                                        [[-16.4688,605.716,173],[0.880315,0.388416,0.250776,0.106249],[-1,2,-2,1],[5921.94,9E+09,9E+09,9E+09,9E+09,9E+09]],
                                        [[-16.4665,606.427,173.764],[0.879525,0.389144,0.251945,0.107365],[-1,2,-2,1],[5919.94,9E+09,9E+09,9E+09,9E+09,9E+09]],
                                        [[-16.4662,607.132,174.535],[0.878733,0.389877,0.253103,0.108461],[-1,2,-2,1],[5917.94,9E+09,9E+09,9E+09,9E+09,9E+09]],
                                        [[-16.463,607.837,175.307],[0.877932,0.390621,0.254258,0.109565],[-1,2,-2,1],[5915.94,9E+09,9E+09,9E+09,9E+09,9E+09]],
                                        [[-16.4608,608.535,176.077],[0.877129,0.391371,0.255402,0.11065],[-1,2,-2,1],[5913.94,9E+09,9E+09,9E+09,9E+09,9E+09]],
                                        [[-16.4544,609.233,176.846],[0.876338,0.392094,0.256543,0.111714],[-1,2,-2,1],[5911.94,9E+09,9E+09,9E+09,9E+09,9E+09]],
                                        [[-16.448,609.934,177.621],[0.875547,0.392822,0.25767,0.112755],[-1,2,-2,1],[5909.94,9E+09,9E+09,9E+09,9E+09,9E+09]],
                                        [[-16.4455,610.629,178.404],[0.874742,0.39359,0.25878,0.113781],[-1,2,-2,1],[5907.94,9E+09,9E+09,9E+09,9E+09,9E+09]],
                                        [[-16.4446,611.323,179.187],[0.873932,0.39437,0.259879,0.114795],[-1,2,-2,1],[5905.94,9E+09,9E+09,9E+09,9E+09,9E+09]],
                                        [[-16.4419,612.013,179.972],[0.87311,0.395177,0.260966,0.115802],[-1,2,-2,1],[5903.94,9E+09,9E+09,9E+09,9E+09,9E+09]],
                                        [[-16.4412,612.703,180.758],[0.872287,0.395996,0.262037,0.116783],[-1,2,-2,1],[5901.94,9E+09,9E+09,9E+09,9E+09,9E+09]],
                                        [[-16.4357,613.389,181.546],[0.871466,0.396828,0.263087,0.117726],[-1,2,-2,1],[5899.94,9E+09,9E+09,9E+09,9E+09,9E+09]],
                                        [[-16.4315,614.073,182.336],[0.870641,0.397685,0.264115,0.118634],[-1,2,-2,1],[5897.94,9E+09,9E+09,9E+09,9E+09,9E+09]],
                                        [[-16.4296,614.755,183.129],[0.869825,0.398544,0.26512,0.119495],[-1,2,-2,1],[5895.94,9E+09,9E+09,9E+09,9E+09,9E+09]],
                                        [[-16.4286,615.436,183.924],[0.869011,0.39942,0.2661,0.120308],[-1,2,-2,1],[5893.94,9E+09,9E+09,9E+09,9E+09,9E+09]],
                                        [[-16.4255,616.116,184.719],[0.868205,0.40029,0.267066,0.12109],[-1,2,-2,1],[5891.94,9E+09,9E+09,9E+09,9E+09,9E+09]],
                                        [[-16.4247,616.797,185.514],[0.867397,0.401171,0.268021,0.121861],[-1,2,-2,1],[5889.94,9E+09,9E+09,9E+09,9E+09,9E+09]],
                                        [[-16.426,617.481,186.317],[0.866592,0.402053,0.268962,0.122605],[-1,2,-2,1],[5887.94,9E+09,9E+09,9E+09,9E+09,9E+09]],
                                        [[-16.4241,618.163,187.124],[0.865786,0.402931,0.2699,0.123348],[-1,2,-2,1],[5885.94,9E+09,9E+09,9E+09,9E+09,9E+09]],
                                        [[-16.4169,618.844,187.93],[0.864989,0.403788,0.270837,0.124084],[-1,2,-2,1],[5883.94,9E+09,9E+09,9E+09,9E+09,9E+09]],
                                        [[-16.4138,619.522,188.739],[0.86419,0.40464,0.271774,0.124824],[-1,2,-2,1],[5881.94,9E+09,9E+09,9E+09,9E+09,9E+09]],
                                        [[-16.4083,620.197,189.55],[0.863399,0.405471,0.27271,0.125558],[-1,2,-2,1],[5879.94,9E+09,9E+09,9E+09,9E+09,9E+09]],
                                        [[-16.4046,620.865,190.357],[0.862604,0.406303,0.273645,0.126297],[-1,2,-2,1],[5877.94,9E+09,9E+09,9E+09,9E+09,9E+09]],
                                        [[-16.3968,621.534,191.171],[0.861814,0.407129,0.27457,0.127018],[-1,2,-2,1],[5875.94,9E+09,9E+09,9E+09,9E+09,9E+09]],
                                        [[-16.3905,622.204,191.985],[0.861029,0.407945,0.275491,0.127729],[-1,2,-2,1],[5873.94,9E+09,9E+09,9E+09,9E+09,9E+09]],
                                        [[-16.3854,622.872,192.8],[0.860247,0.408753,0.276409,0.128433],[-1,2,-2,1],[5871.94,9E+09,9E+09,9E+09,9E+09,9E+09]],
                                        [[-16.3832,623.539,193.617],[0.85946,0.409575,0.277314,0.129126],[-1,2,-2,1],[5869.94,9E+09,9E+09,9E+09,9E+09,9E+09]],
                                        [[-16.3782,624.203,194.438],[0.858671,0.410404,0.27821,0.129811],[-1,2,-2,1],[5867.94,9E+09,9E+09,9E+09,9E+09,9E+09]],
                                        [[-16.3702,624.868,195.256],[0.857885,0.411232,0.279098,0.130482],[-1,2,-2,1],[5865.94,9E+09,9E+09,9E+09,9E+09,9E+09]],
                                        [[-16.36,625.527,196.082],[0.857094,0.412086,0.279965,0.131129],[-1,2,-2,1],[5863.94,9E+09,9E+09,9E+09,9E+09,9E+09]],
                                        [[-16.3521,626.19,196.902],[0.856303,0.412944,0.280822,0.131761],[-1,2,-2,1],[5861.94,9E+09,9E+09,9E+09,9E+09,9E+09]],
                                        [[-16.343,626.851,197.732],[0.855501,0.413827,0.281667,0.132394],[-1,2,-2,1],[5859.94,9E+09,9E+09,9E+09,9E+09,9E+09]],
                                        [[-16.3373,627.513,198.562],[0.85469,0.414724,0.282507,0.133035],[-1,2,-2,1],[5857.94,9E+09,9E+09,9E+09,9E+09,9E+09]],
                                        [[-16.3314,628.172,199.395],[0.853875,0.415619,0.283348,0.133685],[-1,2,-2,1],[5855.94,9E+09,9E+09,9E+09,9E+09,9E+09]],
                                        [[-16.3256,628.826,200.223],[0.853047,0.416519,0.284196,0.134369],[-1,2,-2,1],[5853.94,9E+09,9E+09,9E+09,9E+09,9E+09]],
                                        [[-16.3209,629.482,201.058],[0.852211,0.417405,0.285059,0.135093],[-1,2,-2,1],[5851.94,9E+09,9E+09,9E+09,9E+09,9E+09]],
                                        [[-16.3138,630.136,201.895],[0.851373,0.418283,0.285926,0.135829],[-1,2,-2,1],[5849.94,9E+09,9E+09,9E+09,9E+09,9E+09]],
                                        [[-16.3061,630.787,202.736],[0.85053,0.419166,0.286788,0.136569],[-1,2,-2,1],[5847.94,9E+09,9E+09,9E+09,9E+09,9E+09]],
                                        [[-16.2994,631.434,203.573],[0.849683,0.420043,0.287654,0.137324],[-1,2,-2,1],[5845.94,9E+09,9E+09,9E+09,9E+09,9E+09]],
                                        [[-16.2926,632.082,204.418],[0.848835,0.420916,0.288519,0.138081],[-1,2,-2,1],[5843.94,9E+09,9E+09,9E+09,9E+09,9E+09]],
                                        [[-16.2844,632.728,205.265],[0.847968,0.421816,0.289378,0.138857],[-1,2,-2,1],[5841.94,9E+09,9E+09,9E+09,9E+09,9E+09]],
                                        [[-16.2779,633.376,206.114],[0.847102,0.422713,0.290233,0.139633],[-1,2,-2,1],[5839.94,9E+09,9E+09,9E+09,9E+09,9E+09]],
                                        [[-16.269,634.022,206.966],[0.846219,0.42363,0.291085,0.140426],[-1,2,-2,1],[5837.94,9E+09,9E+09,9E+09,9E+09,9E+09]],
                                        [[-16.254,634.668,207.827],[0.84534,0.42453,0.291941,0.141226],[-1,2,-2,1],[5835.94,9E+09,9E+09,9E+09,9E+09,9E+09]],
                                        [[-16.2422,635.309,208.683],[0.844451,0.425428,0.292804,0.142054],[-1,2,-2,1],[5833.94,9E+09,9E+09,9E+09,9E+09,9E+09]],
                                        [[-16.2264,635.948,209.541],[0.843559,0.426327,0.293663,0.142883],[-1,2,-2,1],[5831.94,9E+09,9E+09,9E+09,9E+09,9E+09]],
                                        [[-16.2095,636.584,210.4],[0.842667,0.427211,0.294528,0.143724],[-1,2,-2,1],[5829.94,9E+09,9E+09,9E+09,9E+09,9E+09]],
                                        [[-16.1954,637.216,211.261],[0.841771,0.428083,0.2954,0.144586],[-1,2,-2,1],[5827.94,9E+09,9E+09,9E+09,9E+09,9E+09]],
                                        [[-16.181,637.839,212.116],[0.840872,0.428941,0.296282,0.145471],[-1,2,-2,1],[5825.94,9E+09,9E+09,9E+09,9E+09,9E+09]],
                                        [[-16.1679,638.455,212.97],[0.83997,0.429778,0.297177,0.14638],[-1,2,-2,1],[5823.94,9E+09,9E+09,9E+09,9E+09,9E+09]],
                                        [[-16.1584,639.071,213.819],[0.839056,0.430609,0.298085,0.147329],[-1,2,-2,1],[5821.94,9E+09,9E+09,9E+09,9E+09,9E+09]],
                                        [[-16.1526,639.686,214.678],[0.838139,0.43142,0.299007,0.148306],[-1,2,-2,1],[5819.94,9E+09,9E+09,9E+09,9E+09,9E+09]],
                                        [[-16.1475,640.301,215.533],[0.837222,0.432196,0.299951,0.149319],[-1,2,-2,1],[5817.94,9E+09,9E+09,9E+09,9E+09,9E+09]],
                                        [[-16.1368,640.913,216.395],[0.836301,0.432942,0.300916,0.150368],[-1,2,-2,1],[5815.94,9E+09,9E+09,9E+09,9E+09,9E+09]],
                                        [[-16.1276,641.526,217.256],[0.83539,0.433649,0.301896,0.151431],[-1,2,-2,1],[5813.94,9E+09,9E+09,9E+09,9E+09,9E+09]],
                                        [[-16.1184,642.14,218.129],[0.834475,0.434361,0.302869,0.152488],[-1,2,-2,1],[5811.94,9E+09,9E+09,9E+09,9E+09,9E+09]],
                                        [[-16.1069,642.748,218.992],[0.833572,0.435048,0.303841,0.153532],[-1,2,-2,1],[5809.94,9E+09,9E+09,9E+09,9E+09,9E+09]],
                                        [[-16.0956,643.35,219.86],[0.832666,0.435728,0.304815,0.154583],[-1,2,-2,1],[5807.94,9E+09,9E+09,9E+09,9E+09,9E+09]],
                                        [[-16.0855,643.953,220.727],[0.831771,0.436383,0.305791,0.155625],[-1,2,-2,1],[5805.94,9E+09,9E+09,9E+09,9E+09,9E+09]],
                                        [[-16.0764,644.555,221.603],[0.83088,0.437017,0.306772,0.156671],[-1,2,-2,1],[5803.94,9E+09,9E+09,9E+09,9E+09,9E+09]],
                                        [[-16.0662,645.154,222.472],[0.829995,0.437631,0.307757,0.157714],[-1,2,-2,1],[5801.94,9E+09,9E+09,9E+09,9E+09,9E+09]],
                                        [[-16.0574,645.75,223.34],[0.829119,0.438233,0.308733,0.158737],[-1,2,-2,1],[5799.94,9E+09,9E+09,9E+09,9E+09,9E+09]],
                                        [[-16.0432,646.341,224.209],[0.828249,0.438818,0.309711,0.159754],[-1,2,-2,1],[5797.94,9E+09,9E+09,9E+09,9E+09,9E+09]],
                                        [[-16.0362,646.93,225.078],[0.827391,0.439394,0.310676,0.16074],[-1,2,-2,1],[5795.94,9E+09,9E+09,9E+09,9E+09,9E+09]],
                                        [[-16.0338,647.518,225.94],[0.826541,0.439972,0.311624,0.161694],[-1,2,-2,1],[5793.94,9E+09,9E+09,9E+09,9E+09,9E+09]],
                                        [[-16.0304,648.102,226.805],[0.825699,0.440542,0.312564,0.162627],[-1,2,-2,1],[5791.94,9E+09,9E+09,9E+09,9E+09,9E+09]],
                                        [[-16.029,648.686,227.678],[0.825273,0.441318,0.312417,0.162967],[-1,2,-2,1],[6236.68,9E+09,9E+09,9E+09,9E+09,9E+09]],
                                        [[-16.0274,649.267,228.552],[0.824444,0.441882,0.313339,0.163861],[-1,2,-2,1],[6236.68,9E+09,9E+09,9E+09,9E+09,9E+09]],
                                        [[-16.0246,649.849,229.427],[0.823612,0.442457,0.314251,0.164747],[-1,2,-2,1],[6236.68,9E+09,9E+09,9E+09,9E+09,9E+09]],
                                        [[-16.0245,650.432,230.308],[0.822787,0.443017,0.31516,0.165623],[-1,2,-2,1],[6236.68,9E+09,9E+09,9E+09,9E+09,9E+09]],
                                        [[-16.0238,651.022,231.193],[0.821962,0.44357,0.316071,0.166503],[-1,2,-2,1],[6236.68,9E+09,9E+09,9E+09,9E+09,9E+09]],
                                        [[-16.02,651.619,232.093],[0.821137,0.444132,0.316968,0.167366],[-1,2,-2,1],[6236.68,9E+09,9E+09,9E+09,9E+09,9E+09]],
                                        [[-16.0079,652.21,232.993],[0.820319,0.44469,0.317856,0.16821],[-1,2,-2,1],[6236.68,9E+09,9E+09,9E+09,9E+09,9E+09]],
                                        [[-15.9949,652.798,233.889],[0.819499,0.445255,0.318735,0.169047],[-1,2,-2,1],[6236.68,9E+09,9E+09,9E+09,9E+09,9E+09]],
                                        [[-15.9855,653.382,234.784],[0.818688,0.445811,0.319607,0.169866],[-1,2,-2,1],[6236.68,9E+09,9E+09,9E+09,9E+09,9E+09]],
                                        [[-15.9753,653.961,235.677],[0.817868,0.446388,0.320465,0.170679],[-1,2,-2,1],[6236.68,9E+09,9E+09,9E+09,9E+09,9E+09]],
                                        [[-15.9659,654.533,236.562],[0.817047,0.446969,0.321316,0.171487],[-1,2,-2,1],[6236.68,9E+09,9E+09,9E+09,9E+09,9E+09]],
                                        [[-15.9573,655.108,237.457],[0.816216,0.447577,0.322152,0.17229],[-1,2,-2,1],[6236.68,9E+09,9E+09,9E+09,9E+09,9E+09]],
                                        [[-15.9494,655.68,238.35],[0.815387,0.448182,0.322983,0.173087],[-1,2,-2,1],[6236.68,9E+09,9E+09,9E+09,9E+09,9E+09]],
                                        [[-15.9432,656.253,239.242],[0.985491,-0.093353,0.141246,-0.0119022],[-1,2,-2,1],[6236.68,9E+09,9E+09,9E+09,9E+09,9E+09]],
                                        [[-15.9337,656.818,240.132],[0.985491,-0.093353,0.141246,-0.0119022],[-1,2,-2,1],[6236.68,9E+09,9E+09,9E+09,9E+09,9E+09]],
                                        [[-15.9252,657.38,241.024],[0.985491,-0.093353,0.141246,-0.0119022],[-1,2,-2,1],[6236.68,9E+09,9E+09,9E+09,9E+09,9E+09]],
                                        [[-15.9178,657.942,241.917],[0.985491,-0.093353,0.141246,-0.0119022],[-1,2,-2,1],[6236.68,9E+09,9E+09,9E+09,9E+09,9E+09]],
                                        [[-15.9128,658.506,242.814],[0.985491,-0.093353,0.141246,-0.0119022],[-1,2,-2,1],[6236.68,9E+09,9E+09,9E+09,9E+09,9E+09]],
                                        [[-15.9043,659.069,243.712],[0.985491,-0.093353,0.141246,-0.0119022],[-1,2,-2,1],[6236.68,9E+09,9E+09,9E+09,9E+09,9E+09]],
                                        [[-15.8949,659.626,244.614],[0.985491,-0.093353,0.141246,-0.0119022],[-1,2,-2,1],[6236.68,9E+09,9E+09,9E+09,9E+09,9E+09]],
                                        [[-15.884,660.185,245.513],[0.985491,-0.093353,0.141246,-0.0119022],[-1,2,-2,1],[6236.68,9E+09,9E+09,9E+09,9E+09,9E+09]],
                                        [[-15.8746,660.737,246.412],[0.985491,-0.093353,0.141246,-0.0119022],[-1,2,-2,1],[6236.68,9E+09,9E+09,9E+09,9E+09,9E+09]],
                                        [[-15.864,661.292,247.315],[0.985491,-0.093353,0.141246,-0.0119022],[-1,2,-2,1],[6236.68,9E+09,9E+09,9E+09,9E+09,9E+09]],
                                        [[-15.8527,661.843,248.221],[0.985491,-0.093353,0.141246,-0.0119022],[-1,2,-2,1],[6236.68,9E+09,9E+09,9E+09,9E+09,9E+09]],
                                        [[-15.843,662.392,249.125],[0.985491,-0.093353,0.141246,-0.0119022],[-1,2,-2,1],[6236.68,9E+09,9E+09,9E+09,9E+09,9E+09]],
                                        [[-15.8348,662.938,250.028],[0.985491,-0.093353,0.141246,-0.0119022],[-1,2,-2,1],[6236.68,9E+09,9E+09,9E+09,9E+09,9E+09]],
                                        [[-15.8269,663.475,250.925],[0.985491,-0.093353,0.141246,-0.0119022],[-1,2,-2,1],[6236.68,9E+09,9E+09,9E+09,9E+09,9E+09]],
                                        [[-15.8195,664.012,251.826],[0.985491,-0.093353,0.141246,-0.0119022],[-1,2,-2,1],[6236.68,9E+09,9E+09,9E+09,9E+09,9E+09]],
                                        [[-15.8093,664.544,252.731],[0.985491,-0.093353,0.141246,-0.0119022],[-1,2,-2,1],[6236.68,9E+09,9E+09,9E+09,9E+09,9E+09]],
                                        [[-15.8028,665.078,253.634],[0.985491,-0.093353,0.141246,-0.0119022],[-1,2,-2,1],[6236.68,9E+09,9E+09,9E+09,9E+09,9E+09]],
                                        [[-15.7448,665.866,254.446],[0.985491,-0.093353,0.141246,-0.0119022],[-1,2,-2,1],[6236.68,9E+09,9E+09,9E+09,9E+09,9E+09]],
                                        [[-15.7745,666.532,255.443],[0.985491,-0.093353,0.141246,-0.0119022],[-1,2,-2,1],[6236.68,9E+09,9E+09,9E+09,9E+09,9E+09]],
                                        [[-15.687,666.936,256.291],[0.985491,-0.093353,0.141246,-0.0119022],[-1,2,-2,1],[6236.68,9E+09,9E+09,9E+09,9E+09,9E+09]],
                                        [[-15.7962,667.567,257.036],[0.985491,-0.093353,0.141246,-0.0119022],[-1,2,-2,1],[6236.68,9E+09,9E+09,9E+09,9E+09,9E+09]],
                                        [[-15.7655,667.961,257.997],[0.985491,-0.093353,0.141246,-0.0119022],[-1,2,-2,1],[6236.68,9E+09,9E+09,9E+09,9E+09,9E+09]],
                                        [[-15.7582,668.439,258.917],[0.985491,-0.093353,0.141246,-0.0119022],[-1,2,-2,1],[6236.68,9E+09,9E+09,9E+09,9E+09,9E+09]],
                                        [[-15.7515,668.992,259.752],[0.985491,-0.093353,0.141246,-0.0119022],[-1,2,-2,1],[6236.68,9E+09,9E+09,9E+09,9E+09,9E+09]],
                                        [[-15.7656,669.642,260.77],[0.985491,-0.093353,0.141246,-0.0119022],[-1,2,-2,1],[6236.68,9E+09,9E+09,9E+09,9E+09,9E+09]],
                                        [[-15.7587,670.18,261.601],[0.985491,-0.093353,0.141246,-0.0119022],[-1,2,-2,1],[6236.68,9E+09,9E+09,9E+09,9E+09,9E+09]],
                                        [[-15.7161,670.57,262.57],[0.985491,-0.093353,0.141246,-0.0119022],[-1,2,-2,1],[6236.68,9E+09,9E+09,9E+09,9E+09,9E+09]],
                                        [[-15.6787,671.123,263.369],[0.985491,-0.093353,0.141246,-0.0119022],[-1,2,-2,1],[6236.68,9E+09,9E+09,9E+09,9E+09,9E+09]],
                                        [[-15.6791,671.49,264.34],[0.985491,-0.093353,0.141246,-0.0119022],[-1,2,-2,1],[6236.68,9E+09,9E+09,9E+09,9E+09,9E+09]],
                                        [[-15.6649,672.148,265.426],[0.985491,-0.093353,0.141246,-0.0119022],[-1,2,-2,1],[6236.68,9E+09,9E+09,9E+09,9E+09,9E+09]],
                                        [[-15.6634,672.552,266.32],[0.985491,-0.093353,0.141246,-0.0119022],[-1,2,-2,1],[6236.68,9E+09,9E+09,9E+09,9E+09,9E+09]],
                                        [[-15.7081,673.113,267.156],[0.985491,-0.093353,0.141246,-0.0119022],[-1,2,-2,1],[6236.68,9E+09,9E+09,9E+09,9E+09,9E+09]],
                                        [[-15.8035,673.64,268.067],[0.985491,-0.093353,0.141246,-0.0119022],[-1,2,-2,1],[6236.68,9E+09,9E+09,9E+09,9E+09,9E+09]],
                                        [[-15.7371,674.137,269.037],[0.985491,-0.093353,0.141246,-0.0119022],[-1,2,-2,1],[6236.68,9E+09,9E+09,9E+09,9E+09,9E+09]],
                                        [[-15.6886,674.748,270.209],[0.985491,-0.093353,0.141246,-0.0119022],[-1,2,-2,1],[6236.68,9E+09,9E+09,9E+09,9E+09,9E+09]],
                                        [[-15.5399,675.156,271.121],[0.985491,-0.093353,0.141246,-0.0119022],[-1,2,-2,1],[6236.68,9E+09,9E+09,9E+09,9E+09,9E+09]],
                                        [[-15.6158,675.69,271.899],[0.985491,-0.093353,0.141246,-0.0119022],[-1,2,-2,1],[6236.68,9E+09,9E+09,9E+09,9E+09,9E+09]],
                                        [[-16.0685,673.406,268.406],[0.77744,0.463066,0.366155,0.216997],[-1,2,-2,1],[5666.45,9E+09,9E+09,9E+09,9E+09,9E+09]],
                                        [[-16.0667,673.912,269.336],[0.776504,0.463677,0.366854,0.21786],[-1,2,-2,1],[5664.45,9E+09,9E+09,9E+09,9E+09,9E+09]],
                                        [[-16.0608,674.413,270.268],[0.775562,0.4643,0.367544,0.218724],[-1,2,-2,1],[5662.45,9E+09,9E+09,9E+09,9E+09,9E+09]],
                                        [[-16.0574,674.912,271.2],[0.774624,0.464915,0.368232,0.219584],[-1,2,-2,1],[5660.45,9E+09,9E+09,9E+09,9E+09,9E+09]],
                                        [[-16.0531,675.409,272.134],[0.773684,0.465512,0.368929,0.220459],[-1,2,-2,1],[5658.45,9E+09,9E+09,9E+09,9E+09,9E+09]],
                                        [[-16.0517,675.907,273.069],[0.772745,0.466095,0.369632,0.221343],[-1,2,-2,1],[5656.45,9E+09,9E+09,9E+09,9E+09,9E+09]],
                                        [[-16.0519,676.4,274.005],[0.771804,0.466665,0.370342,0.222238],[-1,2,-2,1],[5654.45,9E+09,9E+09,9E+09,9E+09,9E+09]],
                                        [[-16.0514,676.893,274.944],[0.770864,0.467217,0.371059,0.223142],[-1,2,-2,1],[5652.45,9E+09,9E+09,9E+09,9E+09,9E+09]],
                                        [[-16.0469,677.385,275.881],[0.769911,0.467761,0.371788,0.224078],[-1,2,-2,1],[5650.45,9E+09,9E+09,9E+09,9E+09,9E+09]],
                                        [[-16.044,677.877,276.826],[0.768946,0.468304,0.372521,0.225035],[-1,2,-2,1],[5648.45,9E+09,9E+09,9E+09,9E+09,9E+09]],
                                        [[-16.0392,678.365,277.773],[0.767988,0.468831,0.373257,0.225989],[-1,2,-2,1],[5646.45,9E+09,9E+09,9E+09,9E+09,9E+09]],
                                        [[-16.036,678.849,278.717],[0.767021,0.469363,0.37399,0.226954],[-1,2,-2,1],[5644.45,9E+09,9E+09,9E+09,9E+09,9E+09]],
                                        [[-16.0322,679.333,279.659],[0.766051,0.469892,0.374724,0.227926],[-1,2,-2,1],[5642.45,9E+09,9E+09,9E+09,9E+09,9E+09]],
                                        [[-16.0278,679.812,280.606],[0.765079,0.470404,0.375466,0.228911],[-1,2,-2,1],[5640.45,9E+09,9E+09,9E+09,9E+09,9E+09]],
                                        [[-16.024,680.293,281.558],[0.764104,0.470915,0.376206,0.229898],[-1,2,-2,1],[5638.45,9E+09,9E+09,9E+09,9E+09,9E+09]],
                                        [[-16.0198,680.773,282.512],[0.763131,0.471429,0.376937,0.230878],[-1,2,-2,1],[5636.45,9E+09,9E+09,9E+09,9E+09,9E+09]],
                                        [[-16.0145,681.251,283.46],[0.762158,0.471947,0.37766,0.231851],[-1,2,-2,1],[5634.45,9E+09,9E+09,9E+09,9E+09,9E+09]],
                                        [[-16.0138,681.724,284.41],[0.761189,0.472469,0.378372,0.23281],[-1,2,-2,1],[5632.45,9E+09,9E+09,9E+09,9E+09,9E+09]],
                                        [[-16.0091,682.195,285.362],[0.760213,0.473002,0.379074,0.233769],[-1,2,-2,1],[5630.45,9E+09,9E+09,9E+09,9E+09,9E+09]],
                                        [[-16.0037,682.663,286.315],[0.759249,0.473515,0.379778,0.23472],[-1,2,-2,1],[5628.45,9E+09,9E+09,9E+09,9E+09,9E+09]],
                                        [[-16.0002,683.132,287.275],[0.758279,0.47404,0.380472,0.235671],[-1,2,-2,1],[5626.45,9E+09,9E+09,9E+09,9E+09,9E+09]],
                                        [[-15.9998,683.601,288.235],[0.75731,0.474559,0.381165,0.236619],[-1,2,-2,1],[5624.45,9E+09,9E+09,9E+09,9E+09,9E+09]],
                                        [[-15.9984,684.066,289.189],[0.756344,0.47506,0.381864,0.237573],[-1,2,-2,1],[5622.45,9E+09,9E+09,9E+09,9E+09,9E+09]],
                                        [[-15.9972,684.528,290.146],[0.755371,0.475548,0.382574,0.238549],[-1,2,-2,1],[5620.45,9E+09,9E+09,9E+09,9E+09,9E+09]],
                                        [[-15.9956,684.993,291.107],[0.754399,0.476012,0.383297,0.239538],[-1,2,-2,1],[5618.45,9E+09,9E+09,9E+09,9E+09,9E+09]],
                                        [[-15.9948,685.455,292.071],[0.753425,0.476466,0.384024,0.240534],[-1,2,-2,1],[5616.45,9E+09,9E+09,9E+09,9E+09,9E+09]],
                                        [[-15.9915,685.91,293.03],[0.752456,0.476913,0.384748,0.241522],[-1,2,-2,1],[5614.45,9E+09,9E+09,9E+09,9E+09,9E+09]],
                                        [[-15.9856,686.361,293.993],[0.751487,0.47735,0.385474,0.242515],[-1,2,-2,1],[5612.45,9E+09,9E+09,9E+09,9E+09,9E+09]],
                                        [[-15.9792,686.815,294.953],[0.750524,0.477787,0.386192,0.243494],[-1,2,-2,1],[5610.45,9E+09,9E+09,9E+09,9E+09,9E+09]],
                                        [[-15.9762,687.264,295.916],[0.749563,0.478218,0.386907,0.24447],[-1,2,-2,1],[5608.45,9E+09,9E+09,9E+09,9E+09,9E+09]],
                                        [[-15.9728,687.713,296.879],[0.748608,0.478635,0.387625,0.245442],[-1,2,-2,1],[5606.45,9E+09,9E+09,9E+09,9E+09,9E+09]],
                                        [[-15.9682,688.157,297.846],[0.747659,0.479026,0.388353,0.246418],[-1,2,-2,1],[5604.45,9E+09,9E+09,9E+09,9E+09,9E+09]],
                                        [[-15.9611,688.602,298.811],[0.746714,0.479407,0.389083,0.24739],[-1,2,-2,1],[5602.45,9E+09,9E+09,9E+09,9E+09,9E+09]],
                                        [[-15.9549,689.045,299.778],[0.74577,0.479767,0.389822,0.248372],[-1,2,-2,1],[5600.45,9E+09,9E+09,9E+09,9E+09,9E+09]],
                                        [[-15.9477,689.484,300.747],[0.744833,0.480109,0.390567,0.249351],[-1,2,-2,1],[5598.45,9E+09,9E+09,9E+09,9E+09,9E+09]],
                                        [[-15.9427,689.92,301.71],[0.743901,0.48041,0.391337,0.250347],[-1,2,-2,1],[5596.45,9E+09,9E+09,9E+09,9E+09,9E+09]],
                                        [[-15.937,690.355,302.679],[0.742968,0.480709,0.392103,0.25134],[-1,2,-2,1],[5594.45,9E+09,9E+09,9E+09,9E+09,9E+09]],
                                        [[-15.9339,690.788,303.649],[0.742046,0.480985,0.392876,0.252328],[-1,2,-2,1],[5592.45,9E+09,9E+09,9E+09,9E+09,9E+09]],
                                        [[-15.9298,691.221,304.618],[0.741122,0.481239,0.393663,0.253332],[-1,2,-2,1],[5590.45,9E+09,9E+09,9E+09,9E+09,9E+09]],
                                        [[-15.9293,691.655,305.587],[0.7402,0.481452,0.394477,0.254355],[-1,2,-2,1],[5588.45,9E+09,9E+09,9E+09,9E+09,9E+09]],
                                        [[-15.9292,692.085,306.557],[0.739277,0.481618,0.395323,0.255407],[-1,2,-2,1],[5586.45,9E+09,9E+09,9E+09,9E+09,9E+09]],
                                        [[-15.9263,692.514,307.521],[0.738364,0.481742,0.396191,0.256467],[-1,2,-2,1],[5584.45,9E+09,9E+09,9E+09,9E+09,9E+09]],
                                        [[-15.9216,692.941,308.493],[0.737456,0.481845,0.397069,0.257528],[-1,1,-2,1],[5582.45,9E+09,9E+09,9E+09,9E+09,9E+09]],
                                        [[-15.9172,693.363,309.467],[0.736562,0.481908,0.397964,0.258584],[-1,1,-2,1],[5580.45,9E+09,9E+09,9E+09,9E+09,9E+09]],
                                        [[-15.9142,693.788,310.44],[0.735675,0.481957,0.398862,0.259633],[-1,1,-2,1],[5578.45,9E+09,9E+09,9E+09,9E+09,9E+09]],
                                        [[-15.9086,694.206,311.41],[0.734792,0.482002,0.399755,0.260673],[-1,1,-2,1],[5576.45,9E+09,9E+09,9E+09,9E+09,9E+09]],
                                        [[-15.9037,694.623,312.379],[0.733929,0.482034,0.400641,0.261681],[-1,1,-2,1],[5574.45,9E+09,9E+09,9E+09,9E+09,9E+09]],
                                        [[-15.9004,695.04,313.347],[0.733084,0.482057,0.401521,0.26266],[-1,1,-2,1],[5572.45,9E+09,9E+09,9E+09,9E+09,9E+09]],
                                        [[-15.8998,695.464,314.319],[0.732249,0.482067,0.402399,0.263625],[-1,1,-2,1],[5570.45,9E+09,9E+09,9E+09,9E+09,9E+09]],
                                        [[-15.8966,695.882,315.293],[0.73142,0.482071,0.403274,0.264579],[-1,1,-2,1],[5568.45,9E+09,9E+09,9E+09,9E+09,9E+09]],
                                        [[-15.8968,696.298,316.268],[0.730612,0.482057,0.404147,0.265505],[-1,1,-2,1],[5566.45,9E+09,9E+09,9E+09,9E+09,9E+09]],
                                        [[-15.8962,696.712,317.237],[0.729816,0.48204,0.405011,0.266408],[-1,1,-2,1],[5564.45,9E+09,9E+09,9E+09,9E+09,9E+09]],
                                        [[-15.8968,697.124,318.204],[0.729028,0.482039,0.405853,0.267281],[-1,1,-2,1],[5562.45,9E+09,9E+09,9E+09,9E+09,9E+09]],
                                        [[-15.8945,697.536,319.179],[0.728241,0.482044,0.406688,0.26815],[-1,1,-2,1],[5560.45,9E+09,9E+09,9E+09,9E+09,9E+09]],
                                        [[-15.8941,697.946,320.155],[0.727464,0.482049,0.407512,0.268995],[-1,1,-2,1],[5558.45,9E+09,9E+09,9E+09,9E+09,9E+09]],
                                        [[-15.8962,698.36,321.128],[0.726692,0.482055,0.40833,0.26983],[-1,1,-2,1],[5556.45,9E+09,9E+09,9E+09,9E+09,9E+09]],
                                        [[-15.8976,698.773,322.102],[0.725921,0.482068,0.409138,0.270656],[-1,1,-2,1],[5554.45,9E+09,9E+09,9E+09,9E+09,9E+09]],
                                        [[-15.9029,699.184,323.07],[0.725166,0.482038,0.409968,0.271479],[-1,1,-2,1],[5552.45,9E+09,9E+09,9E+09,9E+09,9E+09]],
                                        [[-15.9034,699.593,324.039],[0.724399,0.482035,0.41078,0.272302],[-1,1,-2,1],[5550.45,9E+09,9E+09,9E+09,9E+09,9E+09]],
                                        [[-15.9017,700.003,325.014],[0.723643,0.482029,0.411584,0.273107],[-1,1,-2,1],[5548.45,9E+09,9E+09,9E+09,9E+09,9E+09]],
                                        [[-15.8994,700.411,325.991],[0.722893,0.482037,0.412372,0.27389],[-1,1,-2,1],[5546.45,9E+09,9E+09,9E+09,9E+09,9E+09]],
                                        [[-15.8968,700.82,326.967],[0.722152,0.482067,0.413133,0.274642],[-1,1,-2,1],[5544.45,9E+09,9E+09,9E+09,9E+09,9E+09]],
                                        [[-15.8957,701.226,327.943],[0.721418,0.482104,0.413883,0.275378],[-1,1,-2,1],[5542.45,9E+09,9E+09,9E+09,9E+09,9E+09]],
                                        [[-15.8919,701.63,328.913],[0.720677,0.482185,0.4146,0.276097],[-1,1,-2,1],[5540.45,9E+09,9E+09,9E+09,9E+09,9E+09]],
                                        [[-15.8852,702.034,329.889],[0.719947,0.482275,0.415299,0.276791],[-1,1,-2,1],[5538.45,9E+09,9E+09,9E+09,9E+09,9E+09]],
                                        [[-15.8817,702.438,330.867],[0.719219,0.482378,0.415986,0.277472],[-1,1,-2,1],[5536.45,9E+09,9E+09,9E+09,9E+09,9E+09]],
                                        [[-15.8793,702.841,331.844],[0.718488,0.482478,0.416673,0.27816],[-1,1,-2,1],[5534.45,9E+09,9E+09,9E+09,9E+09,9E+09]],
                                        [[-15.8778,703.245,332.821],[0.717754,0.482577,0.417361,0.278854],[-1,1,-2,1],[5532.45,9E+09,9E+09,9E+09,9E+09,9E+09]],
                                        [[-15.8752,703.645,333.801],[0.717017,0.482645,0.418071,0.279567],[-1,1,-2,1],[5530.45,9E+09,9E+09,9E+09,9E+09,9E+09]],
                                        [[-15.8709,704.042,334.781],[0.716271,0.482744,0.418759,0.280277],[-1,1,-2,1],[5528.45,9E+09,9E+09,9E+09,9E+09,9E+09]],
                                        [[-15.87,704.438,335.76],[0.715516,0.482846,0.419447,0.281],[-1,1,-2,1],[5526.45,9E+09,9E+09,9E+09,9E+09,9E+09]],
                                        [[-15.8671,704.833,336.74],[0.714766,0.482971,0.420111,0.281701],[-1,1,-2,1],[5524.45,9E+09,9E+09,9E+09,9E+09,9E+09]],
                                        [[-15.8642,705.23,337.72],[0.714013,0.483103,0.420769,0.282402],[-1,1,-2,1],[5522.45,9E+09,9E+09,9E+09,9E+09,9E+09]],
                                        [[-15.8617,705.629,338.707],[0.71326,0.483239,0.42142,0.2831],[-1,1,-2,1],[5520.45,9E+09,9E+09,9E+09,9E+09,9E+09]],
                                        [[-15.8619,706.026,339.687],[0.712492,0.483398,0.422059,0.283809],[-1,1,-2,1],[5518.45,9E+09,9E+09,9E+09,9E+09,9E+09]],
                                        [[-15.8552,706.417,340.668],[0.711729,0.483526,0.422716,0.284527],[-1,1,-2,1],[5516.45,9E+09,9E+09,9E+09,9E+09,9E+09]],
                                        [[-15.8506,706.804,341.652],[0.710957,0.483669,0.423364,0.28525],[-1,1,-2,1],[5514.45,9E+09,9E+09,9E+09,9E+09,9E+09]],
                                        [[-15.8456,707.196,342.632],[0.710181,0.483818,0.424006,0.285975],[-1,1,-2,1],[5512.45,9E+09,9E+09,9E+09,9E+09,9E+09]],
                                        [[-15.8379,707.588,343.62],[0.709396,0.483997,0.424626,0.286701],[-1,1,-2,1],[5510.45,9E+09,9E+09,9E+09,9E+09,9E+09]],
                                        [[-15.8327,707.976,344.609],[0.708619,0.48414,0.425267,0.287429],[-1,1,-2,1],[5508.45,9E+09,9E+09,9E+09,9E+09,9E+09]],
                                        [[-15.8263,708.36,345.594],[0.707836,0.484296,0.425898,0.288161],[-1,1,-2,1],[5506.45,9E+09,9E+09,9E+09,9E+09,9E+09]],
                                        [[-15.8212,708.747,346.577],[0.707056,0.484479,0.426503,0.288872],[-1,1,-2,1],[5504.45,9E+09,9E+09,9E+09,9E+09,9E+09]],
                                        [[-15.8161,709.132,347.567],[0.706285,0.484676,0.42709,0.289561],[-1,1,-2,1],[5502.45,9E+09,9E+09,9E+09,9E+09,9E+09]],
                                        [[-15.8133,709.517,348.558],[0.70552,0.484883,0.427662,0.290234],[-1,1,-2,1],[5500.45,9E+09,9E+09,9E+09,9E+09,9E+09]],
                                        [[-15.8125,709.903,349.548],[0.704755,0.485104,0.42822,0.290898],[-1,1,-2,1],[5498.45,9E+09,9E+09,9E+09,9E+09,9E+09]],
                                        [[-15.8141,710.291,350.532],[0.70399,0.48533,0.428771,0.29156],[-1,1,-2,1],[5496.45,9E+09,9E+09,9E+09,9E+09,9E+09]],
                                        [[-15.8059,710.668,351.519],[0.703224,0.48558,0.429301,0.292212],[-1,1,-2,1],[5494.45,9E+09,9E+09,9E+09,9E+09,9E+09]],
                                        [[-15.8017,711.048,352.511],[0.702458,0.485859,0.429806,0.292849],[-1,1,-2,1],[5492.45,9E+09,9E+09,9E+09,9E+09,9E+09]],
                                        [[-15.7925,711.425,353.505],[0.701698,0.486143,0.430299,0.293473],[-1,1,-2,1],[5490.45,9E+09,9E+09,9E+09,9E+09,9E+09]],
                                        [[-15.7861,711.803,354.497],[0.700928,0.486471,0.430761,0.294093],[-1,1,-2,1],[5488.45,9E+09,9E+09,9E+09,9E+09,9E+09]],
                                        [[-15.7765,712.177,355.486],[0.700159,0.486804,0.431215,0.294709],[-1,1,-2,1],[5486.45,9E+09,9E+09,9E+09,9E+09,9E+09]],
                                        [[-15.7675,712.547,356.478],[0.699407,0.48713,0.431661,0.295299],[-1,1,-2,1],[5484.45,9E+09,9E+09,9E+09,9E+09,9E+09]],
                                        [[-15.7589,712.922,357.474],[0.698654,0.487461,0.432103,0.295891],[-1,1,-2,1],[5482.45,9E+09,9E+09,9E+09,9E+09,9E+09]],
                                        [[-15.7493,713.293,358.471],[0.697898,0.48781,0.432527,0.296478],[-1,1,-2,1],[5480.45,9E+09,9E+09,9E+09,9E+09,9E+09]],
                                        [[-15.7416,713.659,359.464],[0.697147,0.48814,0.432962,0.29707],[-1,1,-2,1],[5478.45,9E+09,9E+09,9E+09,9E+09,9E+09]],
                                        [[-15.7318,714.025,360.457],[0.696393,0.488474,0.433391,0.297662],[-1,1,-2,1],[5476.45,9E+09,9E+09,9E+09,9E+09,9E+09]],
                                        [[-15.7288,714.396,361.449],[0.69566,0.488793,0.433818,0.298229],[-1,1,-2,1],[5474.45,9E+09,9E+09,9E+09,9E+09,9E+09]],
                                        [[-15.7192,714.765,362.448],[0.694928,0.489113,0.434242,0.298795],[-1,1,-2,1],[5472.45,9E+09,9E+09,9E+09,9E+09,9E+09]],
                                        [[-15.7065,715.126,363.452],[0.694216,0.48944,0.434647,0.299325],[-1,1,-2,1],[5470.45,9E+09,9E+09,9E+09,9E+09,9E+09]],
                                        [[-15.6978,715.488,364.448],[0.693516,0.489745,0.435061,0.299846],[-1,1,-2,1],[5468.45,9E+09,9E+09,9E+09,9E+09,9E+09]],
                                        [[-15.6865,715.847,365.446],[0.69282,0.490052,0.435468,0.300361],[-1,1,-2,1],[5466.45,9E+09,9E+09,9E+09,9E+09,9E+09]],
                                        [[-15.675,716.207,366.443],[0.692123,0.490319,0.435905,0.300898],[-1,1,-2,1],[5464.45,9E+09,9E+09,9E+09,9E+09,9E+09]],
                                        [[-15.6638,716.562,367.441],[0.691419,0.490531,0.436387,0.301471],[-1,1,-2,1],[5462.45,9E+09,9E+09,9E+09,9E+09,9E+09]],
                                        [[-15.6499,716.917,368.442],[0.690718,0.490674,0.436921,0.302074],[-1,1,-2,1],[5460.45,9E+09,9E+09,9E+09,9E+09,9E+09]],
                                        [[-15.6361,717.271,369.442],[0.690018,0.490793,0.43747,0.302685],[-1,1,-2,1],[5458.45,9E+09,9E+09,9E+09,9E+09,9E+09]],
                                        [[-15.6206,717.62,370.445],[0.689296,0.490867,0.438062,0.30335],[-1,1,-2,1],[5456.45,9E+09,9E+09,9E+09,9E+09,9E+09]],
                                        [[-15.6045,717.965,371.45],[0.688575,0.490921,0.438668,0.304024],[-1,1,-2,1],[5454.45,9E+09,9E+09,9E+09,9E+09,9E+09]],
                                        [[-15.5912,718.316,372.452],[0.68786,0.490931,0.439304,0.304708],[-1,1,-2,1],[5452.45,9E+09,9E+09,9E+09,9E+09,9E+09]],
                                        [[-15.5742,718.665,373.455],[0.687132,0.490943,0.439942,0.30541],[-1,1,-2,1],[5450.45,9E+09,9E+09,9E+09,9E+09,9E+09]],
                                        [[-15.5575,719.012,374.458],[0.686416,0.490915,0.440604,0.306111],[-1,1,-2,1],[5448.45,9E+09,9E+09,9E+09,9E+09,9E+09]],
                                        [[-15.5444,719.359,375.461],[0.685696,0.490847,0.441298,0.306833],[-1,1,-2,1],[5446.45,9E+09,9E+09,9E+09,9E+09,9E+09]],
                                        [[-15.5334,719.708,376.463],[0.684969,0.490738,0.442025,0.307584],[-1,1,-2,1],[5444.45,9E+09,9E+09,9E+09,9E+09,9E+09]],
                                        [[-15.5204,720.057,377.465],[0.684232,0.490576,0.442795,0.308372],[-1,1,-2,1],[5442.45,9E+09,9E+09,9E+09,9E+09,9E+09]],
                                        [[-15.5067,720.405,378.467],[0.683475,0.490368,0.44361,0.309211],[-1,1,-2,1],[5440.45,9E+09,9E+09,9E+09,9E+09,9E+09]],
                                        [[-15.4928,720.753,379.47],[0.68272,0.490112,0.444459,0.310065],[-1,1,-2,1],[5438.45,9E+09,9E+09,9E+09,9E+09,9E+09]],
                                        [[-15.4733,721.101,380.473],[0.681971,0.489823,0.44533,0.31092],[-1,1,-2,1],[5436.45,9E+09,9E+09,9E+09,9E+09,9E+09]],
                                        [[-15.4591,721.447,381.477],[0.681219,0.489522,0.446208,0.311782],[-1,1,-2,1],[5434.45,9E+09,9E+09,9E+09,9E+09,9E+09]],
                                        [[-15.4422,721.792,382.48],[0.680463,0.489202,0.447099,0.312654],[-1,1,-2,1],[5432.45,9E+09,9E+09,9E+09,9E+09,9E+09]],
                                        [[-15.4302,722.138,383.48],[0.679714,0.488863,0.448002,0.313523],[-1,1,-2,1],[5430.45,9E+09,9E+09,9E+09,9E+09,9E+09]],
                                        [[-15.4199,722.485,384.476],[0.678955,0.488506,0.448919,0.31441],[-1,1,-2,1],[5428.45,9E+09,9E+09,9E+09,9E+09,9E+09]],
                                        [[-15.406,722.829,385.472],[0.678193,0.488141,0.449841,0.315303],[-1,1,-2,1],[5426.45,9E+09,9E+09,9E+09,9E+09,9E+09]],
                                        [[-15.3944,723.173,386.466],[0.677428,0.487768,0.450767,0.316199],[-1,1,-2,1],[5424.45,9E+09,9E+09,9E+09,9E+09,9E+09]],
                                        [[-15.3875,723.513,387.463],[0.676676,0.487398,0.451683,0.317073],[-1,1,-2,1],[5422.45,9E+09,9E+09,9E+09,9E+09,9E+09]],
                                        [[-15.3759,723.851,388.462],[0.675928,0.487065,0.452566,0.317921],[-1,1,-2,1],[5420.45,9E+09,9E+09,9E+09,9E+09,9E+09]],
                                        [[-15.3637,724.19,389.462],[0.67518,0.486763,0.45342,0.318753],[-1,1,-2,1],[5418.45,9E+09,9E+09,9E+09,9E+09,9E+09]],
                                        [[-15.3519,724.527,390.463],[0.674437,0.486465,0.454267,0.319575],[-1,1,-2,1],[5416.45,9E+09,9E+09,9E+09,9E+09,9E+09]],
                                        [[-15.3395,724.867,391.464],[0.673714,0.486181,0.455092,0.320357],[-1,1,-2,1],[5414.45,9E+09,9E+09,9E+09,9E+09,9E+09]],
                                        [[-15.3306,725.209,392.463],[0.673007,0.485915,0.455894,0.321104],[-1,1,-2,1],[5412.45,9E+09,9E+09,9E+09,9E+09,9E+09]],
                                        [[-15.3232,725.551,393.464],[0.672288,0.485654,0.456695,0.321868],[-1,1,-2,1],[5410.45,9E+09,9E+09,9E+09,9E+09,9E+09]],
                                        [[-15.3168,725.891,394.459],[0.671588,0.485382,0.457495,0.322603],[-1,1,-2,1],[5408.45,9E+09,9E+09,9E+09,9E+09,9E+09]],
                                        [[-15.3141,726.234,395.462],[0.670891,0.48508,0.458314,0.323342],[-1,1,-2,1],[5406.45,9E+09,9E+09,9E+09,9E+09,9E+09]],
                                        [[-15.2991,726.573,396.465],[0.670199,0.484808,0.459107,0.324062],[-1,1,-2,1],[5404.45,9E+09,9E+09,9E+09,9E+09,9E+09]],
                                        [[-15.2868,726.91,397.468],[0.66952,0.484525,0.4599,0.324762],[-1,1,-2,1],[5402.45,9E+09,9E+09,9E+09,9E+09,9E+09]],
                                        [[-15.2765,727.249,398.471],[0.668862,0.484271,0.460661,0.325418],[-1,1,-2,1],[5400.45,9E+09,9E+09,9E+09,9E+09,9E+09]],
                                        [[-15.2636,727.584,399.468],[0.668214,0.48402,0.461413,0.326056],[-1,1,-2,1],[5398.45,9E+09,9E+09,9E+09,9E+09,9E+09]],
                                        [[-15.2512,727.92,400.47],[0.667577,0.483765,0.462164,0.326677],[-1,1,-2,1],[5396.45,9E+09,9E+09,9E+09,9E+09,9E+09]],
                                        [[-15.2418,728.252,401.473],[0.666944,0.483507,0.462912,0.32729],[-1,1,-2,1],[5394.45,9E+09,9E+09,9E+09,9E+09,9E+09]],
                                        [[-15.2297,728.588,402.474],[0.666312,0.483244,0.463663,0.327903],[-1,1,-2,1],[5392.45,9E+09,9E+09,9E+09,9E+09,9E+09]],
                                        [[-15.2199,728.921,403.478],[0.665699,0.482978,0.464408,0.328486],[-1,1,-2,1],[5390.45,9E+09,9E+09,9E+09,9E+09,9E+09]],
                                        [[-15.2053,729.257,404.484],[0.665099,0.482718,0.465141,0.329045],[-1,1,-2,1],[5388.45,9E+09,9E+09,9E+09,9E+09,9E+09]],
                                        [[-15.1891,729.589,405.493],[0.664495,0.482423,0.465901,0.329624],[-1,1,-2,1],[5386.45,9E+09,9E+09,9E+09,9E+09,9E+09]],
                                        [[-15.1752,729.919,406.505],[0.663893,0.482126,0.466656,0.330203],[-1,1,-2,1],[5384.45,9E+09,9E+09,9E+09,9E+09,9E+09]],
                                        [[-15.1619,730.254,407.517],[0.663285,0.481841,0.467401,0.330785],[-1,1,-2,1],[5382.45,9E+09,9E+09,9E+09,9E+09,9E+09]],
                                        [[-15.1469,730.592,408.526],[0.662675,0.481524,0.468171,0.331379],[-1,1,-2,1],[5380.45,9E+09,9E+09,9E+09,9E+09,9E+09]],
                                        [[-15.1327,730.933,409.534],[0.662066,0.481202,0.468943,0.331973],[-1,1,-2,1],[5378.45,9E+09,9E+09,9E+09,9E+09,9E+09]],
                                        [[-15.1232,731.269,410.539],[0.661467,0.480853,0.46973,0.332558],[-1,1,-2,1],[5376.45,9E+09,9E+09,9E+09,9E+09,9E+09]],
                                        [[-15.1069,731.606,411.543],[0.660869,0.480478,0.470536,0.333149],[-1,1,-2,1],[5374.45,9E+09,9E+09,9E+09,9E+09,9E+09]],
                                        [[-15.0984,731.944,412.546],[0.660258,0.480074,0.471367,0.333768],[-1,1,-2,1],[5372.45,9E+09,9E+09,9E+09,9E+09,9E+09]],
                                        [[-15.0826,732.276,413.551],[0.659617,0.479594,0.472264,0.334456],[-1,1,-2,1],[5370.45,9E+09,9E+09,9E+09,9E+09,9E+09]],
                                        [[-15.0702,732.611,414.555],[0.658981,0.479095,0.473173,0.335141],[-1,1,-2,1],[5368.45,9E+09,9E+09,9E+09,9E+09,9E+09]],
                                        [[-15.0566,732.946,415.566],[0.658331,0.478558,0.474113,0.335855],[-1,1,-2,1],[5366.45,9E+09,9E+09,9E+09,9E+09,9E+09]],
                                        [[-15.0441,733.282,416.569],[0.657686,0.478009,0.475059,0.336564],[-1,1,-2,1],[5364.45,9E+09,9E+09,9E+09,9E+09,9E+09]],
                                        [[-15.0354,733.619,417.571],[0.657042,0.477445,0.476014,0.337272],[-1,1,-2,1],[5362.45,9E+09,9E+09,9E+09,9E+09,9E+09]],
                                        [[-15.0232,733.952,418.575],[0.6564,0.476866,0.476976,0.337982],[-1,1,-2,1],[5360.45,9E+09,9E+09,9E+09,9E+09,9E+09]],
                                        [[-15.0104,734.283,419.58],[0.655747,0.476269,0.477948,0.338717],[-1,1,-2,1],[5358.45,9E+09,9E+09,9E+09,9E+09,9E+09]],
                                        [[-14.9969,734.617,420.591],[0.655105,0.475685,0.4789,0.339436],[-1,1,-2,1],[5356.45,9E+09,9E+09,9E+09,9E+09,9E+09]],
                                        [[-14.9809,734.949,421.597],[0.654473,0.475099,0.479842,0.340144],[-1,1,-2,1],[5354.45,9E+09,9E+09,9E+09,9E+09,9E+09]],
                                        [[-14.9707,735.289,422.6],[0.653848,0.474525,0.480766,0.340842],[-1,1,-2,1],[5352.45,9E+09,9E+09,9E+09,9E+09,9E+09]],
                                        [[-14.9603,735.625,423.604],[0.653234,0.473923,0.4817,0.341537],[-1,1,-2,1],[5350.45,9E+09,9E+09,9E+09,9E+09,9E+09]],
                                        [[-14.9478,735.957,424.609],[0.652613,0.47333,0.48262,0.342246],[-1,1,-2,1],[5348.45,9E+09,9E+09,9E+09,9E+09,9E+09]],
                                        [[-14.941,736.292,425.612],[0.652004,0.472732,0.483533,0.342945],[-1,1,-2,1],[5346.45,9E+09,9E+09,9E+09,9E+09,9E+09]],
                                        [[-14.9303,736.629,426.616],[0.651412,0.472157,0.484414,0.343619],[-1,1,-2,1],[5344.45,9E+09,9E+09,9E+09,9E+09,9E+09]],
                                        [[-14.917,736.969,427.619],[0.650851,0.471586,0.485272,0.344252],[-1,1,-2,1],[5342.45,9E+09,9E+09,9E+09,9E+09,9E+09]],
                                        [[-14.9037,737.304,428.623],[0.650311,0.471004,0.486125,0.344869],[-1,1,-2,1],[5340.45,9E+09,9E+09,9E+09,9E+09,9E+09]],
                                        [[-14.8931,737.64,429.628],[0.649806,0.470454,0.486933,0.34543],[-1,1,-2,1],[5338.45,9E+09,9E+09,9E+09,9E+09,9E+09]],
                                        [[-14.8881,737.98,430.637],[0.649316,0.469874,0.487749,0.345988],[-1,1,-2,1],[5336.45,9E+09,9E+09,9E+09,9E+09,9E+09]],
                                        [[-14.8805,738.323,431.639],[0.648853,0.469313,0.488533,0.346512],[-1,1,-2,1],[5334.45,9E+09,9E+09,9E+09,9E+09,9E+09]],
                                        [[-14.8768,738.663,432.642],[0.648399,0.468764,0.489296,0.347029],[-1,1,-2,1],[5332.45,9E+09,9E+09,9E+09,9E+09,9E+09]],
                                        [[-14.8641,739,433.646],[0.647972,0.468242,0.49002,0.347508],[-1,1,-2,1],[5330.45,9E+09,9E+09,9E+09,9E+09,9E+09]],
                                        [[-14.8549,739.339,434.65],[0.64758,0.467761,0.490695,0.347934],[-1,1,-2,1],[5328.45,9E+09,9E+09,9E+09,9E+09,9E+09]],
                                        [[-14.8463,739.68,435.66],[0.647205,0.467298,0.491342,0.348341],[-1,1,-2,1],[5326.45,9E+09,9E+09,9E+09,9E+09,9E+09]],
                                        [[-14.8402,740.019,436.664],[0.646852,0.466879,0.491941,0.348714],[-1,1,-2,1],[5324.45,9E+09,9E+09,9E+09,9E+09,9E+09]],
                                        [[-14.8279,740.354,437.67],[0.646503,0.466494,0.492502,0.349082],[-1,1,-2,1],[5322.45,9E+09,9E+09,9E+09,9E+09,9E+09]],
                                        [[-14.8158,740.692,438.678],[0.646176,0.466102,0.493055,0.349432],[-1,1,-2,1],[5320.45,9E+09,9E+09,9E+09,9E+09,9E+09]],
                                        [[-14.807,741.033,439.684],[0.64587,0.465788,0.493534,0.349739],[-1,1,-2,1],[5318.45,9E+09,9E+09,9E+09,9E+09,9E+09]],
                                        [[-14.8053,741.382,440.696],[0.645592,0.465499,0.493979,0.350011],[-1,1,-2,1],[5316.45,9E+09,9E+09,9E+09,9E+09,9E+09]],
                                        [[-14.8011,741.728,441.704],[0.645326,0.46522,0.494403,0.350271],[-1,1,-2,1],[5314.45,9E+09,9E+09,9E+09,9E+09,9E+09]],
                                        [[-14.7951,742.072,442.713],[0.645071,0.464959,0.494804,0.350521],[-1,1,-2,1],[5312.45,9E+09,9E+09,9E+09,9E+09,9E+09]],
                                        [[-14.7863,742.413,443.725],[0.644819,0.464712,0.495185,0.350776],[-1,1,-2,1],[5310.45,9E+09,9E+09,9E+09,9E+09,9E+09]],
                                        [[-14.7769,742.76,444.737],[0.644598,0.464495,0.495528,0.350985],[-1,1,-2,1],[5308.45,9E+09,9E+09,9E+09,9E+09,9E+09]],
                                        [[-14.7682,743.111,445.747],[0.644402,0.464337,0.495813,0.351152],[-1,1,-2,1],[5306.45,9E+09,9E+09,9E+09,9E+09,9E+09]],
                                        [[-14.7566,743.457,446.755],[0.644226,0.4642,0.49607,0.351292],[-1,1,-2,1],[5304.45,9E+09,9E+09,9E+09,9E+09,9E+09]],
                                        [[-14.7514,743.804,447.76],[0.644066,0.46408,0.496304,0.351413],[-1,1,-2,1],[5302.45,9E+09,9E+09,9E+09,9E+09,9E+09]],
                                        [[-14.7444,744.148,448.763],[0.643887,0.463947,0.496546,0.351574],[-1,1,-2,1],[5300.45,9E+09,9E+09,9E+09,9E+09,9E+09]],
                                        [[-14.7396,744.494,449.764],[0.643707,0.463803,0.496791,0.351748],[-1,1,-2,1],[5298.45,9E+09,9E+09,9E+09,9E+09,9E+09]],
                                        [[-14.7297,744.836,450.764],[0.643516,0.463643,0.497046,0.351948],[-1,1,-2,1],[5296.45,9E+09,9E+09,9E+09,9E+09,9E+09]],
                                        [[-14.7158,745.172,451.758],[0.643338,0.463519,0.497266,0.352126],[-1,1,-2,1],[5294.45,9E+09,9E+09,9E+09,9E+09,9E+09]],
                                        [[-14.7047,745.509,452.757],[0.643162,0.463408,0.497471,0.352304],[-1,1,-2,1],[5292.45,9E+09,9E+09,9E+09,9E+09,9E+09]],
                                        [[-14.6924,745.846,453.758],[0.642975,0.463318,0.497661,0.352496],[-1,1,-2,1],[5290.45,9E+09,9E+09,9E+09,9E+09,9E+09]],
                                        [[-14.6861,746.185,454.759],[0.642782,0.463218,0.497856,0.352704],[-1,1,-2,1],[5288.45,9E+09,9E+09,9E+09,9E+09,9E+09]],
                                        [[-14.6833,746.526,455.761],[0.64261,0.463147,0.498021,0.352877],[-1,1,-2,1],[5286.45,9E+09,9E+09,9E+09,9E+09,9E+09]],
                                        [[-14.6709,746.863,456.757],[0.642449,0.463123,0.498146,0.353024],[-1,1,-2,1],[5284.45,9E+09,9E+09,9E+09,9E+09,9E+09]],
                                        [[-14.6591,747.201,457.76],[0.642305,0.463106,0.49826,0.353148],[-1,1,-2,1],[5282.45,9E+09,9E+09,9E+09,9E+09,9E+09]],
                                        [[-14.6527,747.544,458.762],[0.64216,0.463076,0.498382,0.353278],[-1,1,-2,1],[5280.45,9E+09,9E+09,9E+09,9E+09,9E+09]],
                                        [[-14.6476,747.886,459.762],[0.642028,0.463063,0.498488,0.353386],[-1,1,-2,1],[5278.45,9E+09,9E+09,9E+09,9E+09,9E+09]],
                                        [[-14.6398,748.228,460.762],[0.641901,0.463037,0.498602,0.353491],[-1,1,-2,1],[5276.45,9E+09,9E+09,9E+09,9E+09,9E+09]],
                                        [[-14.6269,748.564,461.755],[0.641774,0.463012,0.498714,0.353595],[-1,1,-2,1],[5274.45,9E+09,9E+09,9E+09,9E+09,9E+09]],
                                        [[-14.6138,748.899,462.753],[0.641662,0.462978,0.498829,0.353682],[-1,1,-2,1],[5272.45,9E+09,9E+09,9E+09,9E+09,9E+09]],
                                        [[-14.607,749.238,463.751],[0.641564,0.462945,0.498939,0.353748],[-1,1,-2,1],[5270.45,9E+09,9E+09,9E+09,9E+09,9E+09]],
                                        [[-14.5986,749.578,464.746],[0.641492,0.462915,0.499039,0.353777],[-1,1,-2,1],[5268.45,9E+09,9E+09,9E+09,9E+09,9E+09]],
                                        [[-14.5963,749.916,465.74],[0.64143,0.462881,0.49914,0.353791],[-1,1,-2,1],[5266.45,9E+09,9E+09,9E+09,9E+09,9E+09]],
                                        [[-14.5925,750.252,466.737],[0.641372,0.462806,0.49927,0.353811],[-1,1,-2,1],[5264.45,9E+09,9E+09,9E+09,9E+09,9E+09]],
                                        [[-14.5868,750.59,467.736],[0.64131,0.462701,0.499423,0.353844],[-1,1,-2,1],[5262.45,9E+09,9E+09,9E+09,9E+09,9E+09]],
                                        [[-14.5784,750.925,468.738],[0.641259,0.462587,0.49958,0.353863],[-1,1,-2,1],[5260.45,9E+09,9E+09,9E+09,9E+09,9E+09]],
                                        [[-14.5714,751.261,469.742],[0.641227,0.462514,0.499704,0.353844],[-1,1,-2,1],[5258.45,9E+09,9E+09,9E+09,9E+09,9E+09]],
                                        [[-14.565,751.599,470.748],[0.641198,0.462456,0.499816,0.353814],[-1,1,-2,1],[5256.45,9E+09,9E+09,9E+09,9E+09,9E+09]],
                                        [[-14.5594,751.94,471.756],[0.641183,0.462416,0.499912,0.353755],[-1,1,-2,1],[5254.45,9E+09,9E+09,9E+09,9E+09,9E+09]],
                                        [[-14.5488,752.284,472.772],[0.64117,0.462379,0.500008,0.353694],[-1,1,-2,1],[5252.45,9E+09,9E+09,9E+09,9E+09,9E+09]],
                                        [[-14.5375,752.624,473.783],[0.641148,0.462295,0.50014,0.353655],[-1,1,-2,1],[5250.45,9E+09,9E+09,9E+09,9E+09,9E+09]],
                                        [[-14.527,752.97,474.792],[0.641138,0.462239,0.500251,0.353591],[-1,1,-2,1],[5248.45,9E+09,9E+09,9E+09,9E+09,9E+09]],
                                        [[-14.5148,753.315,475.801],[0.641146,0.462176,0.500364,0.3535],[-1,1,-2,1],[5246.45,9E+09,9E+09,9E+09,9E+09,9E+09]],
                                        [[-14.4974,753.657,476.811],[0.641155,0.462073,0.500507,0.353414],[-1,1,-2,1],[5244.45,9E+09,9E+09,9E+09,9E+09,9E+09]],
                                        [[-14.4868,754.002,477.82],[0.641167,0.461953,0.500664,0.353328],[-1,1,-2,1],[5242.45,9E+09,9E+09,9E+09,9E+09,9E+09]],
                                        [[-14.4779,754.348,478.828],[0.641188,0.461814,0.500834,0.35323],[-1,1,-2,1],[5240.45,9E+09,9E+09,9E+09,9E+09,9E+09]],
                                        [[-14.4685,754.694,479.834],[0.641225,0.461663,0.50101,0.353109],[-1,1,-2,1],[5238.45,9E+09,9E+09,9E+09,9E+09,9E+09]],
                                        [[-14.4565,755.04,480.84],[0.641271,0.461506,0.501191,0.352977],[-1,1,-2,1],[5236.45,9E+09,9E+09,9E+09,9E+09,9E+09]],
                                        [[-14.4449,755.386,481.846],[0.641297,0.461309,0.501405,0.352882],[-1,1,-2,1],[5234.45,9E+09,9E+09,9E+09,9E+09,9E+09]],
                                        [[-14.4305,755.732,482.85],[0.641341,0.46107,0.501648,0.352768],[-1,1,-2,1],[5232.45,9E+09,9E+09,9E+09,9E+09,9E+09]],
                                        [[-14.4243,756.082,483.851],[0.641385,0.460792,0.501922,0.352664],[-1,1,-2,1],[5230.45,9E+09,9E+09,9E+09,9E+09,9E+09]],
                                        [[-14.4155,756.429,484.847],[0.641411,0.460484,0.502222,0.352589],[-1,1,-2,1],[5228.45,9E+09,9E+09,9E+09,9E+09,9E+09]],
                                        [[-14.4062,756.771,485.842],[0.641434,0.460143,0.502551,0.352524],[-1,1,-2,1],[5226.45,9E+09,9E+09,9E+09,9E+09,9E+09]],
                                        [[-14.3916,757.109,486.839],[0.641454,0.459784,0.502894,0.352468],[-1,1,-2,1],[5224.45,9E+09,9E+09,9E+09,9E+09,9E+09]],
                                        [[-14.3807,757.449,487.838],[0.641469,0.459409,0.503252,0.352418],[-1,1,-2,1],[5222.45,9E+09,9E+09,9E+09,9E+09,9E+09]],
                                        [[-14.3684,757.791,488.831],[0.641481,0.458999,0.503637,0.35238],[-1,1,-2,1],[5220.45,9E+09,9E+09,9E+09,9E+09,9E+09]],
                                        [[-14.3548,758.136,489.831],[0.641502,0.458565,0.50404,0.352331],[-1,1,-2,1],[5218.45,9E+09,9E+09,9E+09,9E+09,9E+09]],
                                        [[-14.3461,758.486,490.829],[0.641539,0.458121,0.504446,0.352258],[-1,1,-2,1],[5216.45,9E+09,9E+09,9E+09,9E+09,9E+09]],
                                        [[-14.3326,758.837,491.828],[0.641596,0.457669,0.504856,0.352156],[-1,1,-2,1],[5214.45,9E+09,9E+09,9E+09,9E+09,9E+09]],
                                        [[-14.3211,759.188,492.828],[0.641671,0.457178,0.50529,0.352035],[-1,1,-2,1],[5212.45,9E+09,9E+09,9E+09,9E+09,9E+09]],
                                        [[-14.3127,759.541,493.828],[0.641755,0.456669,0.505736,0.351902],[-1,1,-2,1],[5210.45,9E+09,9E+09,9E+09,9E+09,9E+09]],
                                        [[-14.2993,759.896,494.825],[0.641871,0.456159,0.506175,0.35172],[-1,1,-2,1],[5208.45,9E+09,9E+09,9E+09,9E+09,9E+09]],
                                        [[-14.2865,760.25,495.822],[0.64201,0.455638,0.506618,0.351505],[-1,1,-2,1],[5206.45,9E+09,9E+09,9E+09,9E+09,9E+09]],
                                        [[-14.2771,760.606,496.818],[0.642163,0.455088,0.507077,0.351275],[-1,1,-2,1],[5204.45,9E+09,9E+09,9E+09,9E+09,9E+09]],
                                        [[-14.2693,760.963,497.81],[0.642325,0.45452,0.507546,0.351038],[-1,1,-2,1],[5202.45,9E+09,9E+09,9E+09,9E+09,9E+09]],
                                        [[-14.2657,761.324,498.807],[0.642506,0.453904,0.508043,0.350783],[-1,1,-2,1],[5200.45,9E+09,9E+09,9E+09,9E+09,9E+09]],
                                        [[-14.2557,761.687,499.797],[0.642698,0.453272,0.508548,0.350518],[-1,1,-2,1],[5198.45,9E+09,9E+09,9E+09,9E+09,9E+09]],
                                        [[-14.2431,762.046,500.789],[0.642915,0.452644,0.509041,0.350215],[-1,1,-2,1],[5196.45,9E+09,9E+09,9E+09,9E+09,9E+09]],
                                        [[-14.2334,762.406,501.78],[0.643154,0.451964,0.509565,0.349893],[-1,1,-2,1],[5194.45,9E+09,9E+09,9E+09,9E+09,9E+09]],
                                        [[-14.2227,762.773,502.777],[0.643413,0.451292,0.510074,0.349542],[-1,1,-2,1],[5192.45,9E+09,9E+09,9E+09,9E+09,9E+09]],
                                        [[-14.2127,763.139,503.774],[0.643687,0.450607,0.510586,0.349172],[-1,1,-2,1],[5190.45,9E+09,9E+09,9E+09,9E+09,9E+09]],
                                        [[-14.2011,763.507,504.768],[0.643981,0.449927,0.511087,0.348775],[-1,1,-2,1],[5188.45,9E+09,9E+09,9E+09,9E+09,9E+09]],
                                        [[-14.1905,763.879,505.764],[0.644269,0.449243,0.511588,0.34839],[-1,1,-2,1],[5186.45,9E+09,9E+09,9E+09,9E+09,9E+09]],
                                        [[-14.1751,764.255,506.762],[0.644561,0.448547,0.512093,0.348005],[-1,1,-2,1],[5184.45,9E+09,9E+09,9E+09,9E+09,9E+09]],
                                        [[-14.1608,764.637,507.758],[0.644865,0.44785,0.512591,0.347605],[-1,1,-2,1],[5182.45,9E+09,9E+09,9E+09,9E+09,9E+09]],
                                        [[-14.1459,765.02,508.758],[0.645168,0.44714,0.513096,0.347213],[-1,1,-2,1],[5180.45,9E+09,9E+09,9E+09,9E+09,9E+09]],
                                        [[-14.1349,765.406,509.756],[0.645482,0.446443,0.513584,0.346805],[-1,1,-2,1],[5178.45,9E+09,9E+09,9E+09,9E+09,9E+09]],
                                        [[-14.1246,765.792,510.746],[0.645791,0.44573,0.514083,0.346407],[-1,1,-2,1],[5176.45,9E+09,9E+09,9E+09,9E+09,9E+09]],
                                        [[-14.1127,766.179,511.734],[0.646097,0.445002,0.51459,0.346021],[-1,1,-2,1],[5174.45,9E+09,9E+09,9E+09,9E+09,9E+09]],
                                        [[-14.0978,766.566,512.722],[0.646412,0.444263,0.515096,0.345626],[-1,1,-2,1],[5172.45,9E+09,9E+09,9E+09,9E+09,9E+09]],
                                        [[-14.0851,766.959,513.714],[0.646728,0.443535,0.51559,0.345233],[-1,1,-2,1],[5170.45,9E+09,9E+09,9E+09,9E+09,9E+09]],
                                        [[-14.0735,767.354,514.697],[0.64704,0.442793,0.51609,0.344855],[-1,1,-2,1],[5168.45,9E+09,9E+09,9E+09,9E+09,9E+09]],
                                        [[-14.0662,767.748,515.68],[0.647342,0.442046,0.516589,0.344498],[-1,1,-2,1],[5166.45,9E+09,9E+09,9E+09,9E+09,9E+09]],
                                        [[-14.0568,768.142,516.665],[0.647616,0.441262,0.517116,0.344198],[-1,1,-2,1],[5164.45,9E+09,9E+09,9E+09,9E+09,9E+09]],
                                        [[-14.0437,768.541,517.648],[0.647895,0.440463,0.517646,0.343899],[-1,1,-2,1],[5162.45,9E+09,9E+09,9E+09,9E+09,9E+09]],
                                        [[-14.0313,768.946,518.635],[0.64817,0.439694,0.518151,0.343604],[-1,1,-2,1],[5160.45,9E+09,9E+09,9E+09,9E+09,9E+09]],
                                        [[-14.0137,769.348,519.617],[0.648437,0.438938,0.518642,0.343325],[-1,1,-2,1],[5158.45,9E+09,9E+09,9E+09,9E+09,9E+09]],
                                        [[-13.9997,769.75,520.598],[0.648708,0.438192,0.519121,0.343045],[-1,1,-2,1],[5156.45,9E+09,9E+09,9E+09,9E+09,9E+09]],
                                        [[-13.9877,770.156,521.579],[0.648956,0.43746,0.519588,0.342802],[-1,1,-2,1],[5154.45,9E+09,9E+09,9E+09,9E+09,9E+09]],
                                        [[-13.9793,770.566,522.56],[0.6492,0.436737,0.520044,0.34257],[-1,1,-2,1],[5152.45,9E+09,9E+09,9E+09,9E+09,9E+09]],
                                        [[-13.9719,770.974,523.533],[0.649422,0.436023,0.520496,0.342371],[-1,1,-2,1],[5154.45,9E+09,9E+09,9E+09,9E+09,9E+09]],
                                        [[-13.9618,771.385,524.512],[0.649648,0.435319,0.520939,0.342165],[-1,1,-2,1],[5152.45,9E+09,9E+09,9E+09,9E+09,9E+09]],
                                        [[-13.9524,771.797,525.491],[0.649866,0.434633,0.521371,0.341967],[-1,1,-2,1],[5154.45,9E+09,9E+09,9E+09,9E+09,9E+09]],
                                        [[-13.9408,772.211,526.469],[0.650081,0.433975,0.521781,0.341766],[-1,1,-2,1],[5152.45,9E+09,9E+09,9E+09,9E+09,9E+09]],
                                        [[-13.934,772.625,527.448],[0.650297,0.433349,0.522169,0.341557],[-1,1,-2,1],[5150.45,9E+09,9E+09,9E+09,9E+09,9E+09]],
                                        [[-13.9249,773.043,528.427],[0.650516,0.432727,0.522553,0.341344],[-1,1,-2,1],[5152.45,9E+09,9E+09,9E+09,9E+09,9E+09]],
                                        [[-13.918,773.467,529.406],[0.650731,0.432138,0.522913,0.341128],[-1,1,-2,1],[5150.45,9E+09,9E+09,9E+09,9E+09,9E+09]],
                                        [[-13.9101,773.889,530.385],[0.650945,0.431575,0.523255,0.340906],[-1,1,-2,1],[5152.45,9E+09,9E+09,9E+09,9E+09,9E+09]],
                                        [[-13.9039,774.315,531.367],[0.651163,0.431031,0.523583,0.340677],[-1,1,-2,1],[5150.45,9E+09,9E+09,9E+09,9E+09,9E+09]],
                                        [[-13.8961,774.742,532.35],[0.651391,0.430485,0.523909,0.34043],[-1,1,-2,1],[5152.45,9E+09,9E+09,9E+09,9E+09,9E+09]],
                                        [[-13.8937,775.17,533.336],[0.65161,0.429961,0.524221,0.340191],[-1,1,-2,1],[5150.45,9E+09,9E+09,9E+09,9E+09,9E+09]],
                                        [[-13.8862,775.598,534.315],[0.65183,0.429452,0.524522,0.339948],[-1,1,-2,1],[5152.45,9E+09,9E+09,9E+09,9E+09,9E+09]],
                                        [[-13.8771,776.024,535.294],[0.652047,0.428973,0.524803,0.339703],[-1,1,-2,1],[5150.45,9E+09,9E+09,9E+09,9E+09,9E+09]],
                                        [[-13.869,776.452,536.27],[0.652274,0.428501,0.525076,0.339442],[-1,1,-2,1],[5152.45,9E+09,9E+09,9E+09,9E+09,9E+09]],
                                        [[-13.8595,776.885,537.247],[0.652522,0.428077,0.525312,0.339134],[-1,1,-2,1],[5150.45,9E+09,9E+09,9E+09,9E+09,9E+09]],
                                        [[-13.8554,777.315,538.225],[0.652787,0.427688,0.52552,0.338793],[-1,1,-2,1],[5152.45,9E+09,9E+09,9E+09,9E+09,9E+09]],
                                        [[-13.8495,777.744,539.198],[0.653059,0.427298,0.525727,0.338439],[-1,1,-2,1],[5150.45,9E+09,9E+09,9E+09,9E+09,9E+09]],
                                        [[-13.8456,778.177,540.169],[0.653327,0.426906,0.525936,0.338092],[-1,1,-2,1],[5152.45,9E+09,9E+09,9E+09,9E+09,9E+09]],
                                        [[-13.8394,778.613,541.14],[0.653594,0.426498,0.526155,0.33775],[-1,1,-2,1],[5150.45,9E+09,9E+09,9E+09,9E+09,9E+09]],
                                        [[-13.8344,779.05,542.115],[0.653882,0.426079,0.526377,0.337375],[-1,1,-2,1],[5152.45,9E+09,9E+09,9E+09,9E+09,9E+09]],
                                        [[-13.8271,779.487,543.089],[0.654167,0.425676,0.526589,0.337001],[-1,1,-2,1],[5154.45,9E+09,9E+09,9E+09,9E+09,9E+09]],
                                        [[-13.8152,779.922,544.064],[0.654465,0.42529,0.526786,0.336601],[-1,1,-2,1],[5152.45,9E+09,9E+09,9E+09,9E+09,9E+09]],
                                        [[-13.8063,780.358,545.031],[0.654768,0.424894,0.526988,0.336194],[-1,1,-2,1],[5154.45,9E+09,9E+09,9E+09,9E+09,9E+09]],
                                        [[-13.7959,780.795,545.997],[0.655088,0.424506,0.527181,0.335758],[-1,1,-2,1],[5152.45,9E+09,9E+09,9E+09,9E+09,9E+09]],
                                        [[-13.7893,781.236,546.963],[0.655423,0.424104,0.527381,0.3353],[-1,1,-2,1],[5154.45,9E+09,9E+09,9E+09,9E+09,9E+09]],
                                        [[-13.7808,781.68,547.933],[0.655763,0.423687,0.527588,0.334836],[-1,1,-2,1],[5152.45,9E+09,9E+09,9E+09,9E+09,9E+09]],
                                        [[-13.7728,782.124,548.902],[0.656117,0.423243,0.52781,0.334353],[-1,1,-2,1],[5154.45,9E+09,9E+09,9E+09,9E+09,9E+09]],
                                        [[-13.7618,782.564,549.862],[0.656483,0.422779,0.528043,0.333854],[-1,1,-2,1],[5152.45,9E+09,9E+09,9E+09,9E+09,9E+09]],
                                        [[-13.7514,783.004,550.82],[0.656852,0.422288,0.528292,0.333355],[-1,1,-2,1],[5154.45,9E+09,9E+09,9E+09,9E+09,9E+09]],
                                        [[-13.7433,783.446,551.773],[0.657233,0.421764,0.528561,0.332843],[-1,1,-2,1],[5156.45,9E+09,9E+09,9E+09,9E+09,9E+09]],
                                        [[-13.7352,783.889,552.732],[0.657618,0.421219,0.528841,0.332325],[-1,1,-2,1],[5154.45,9E+09,9E+09,9E+09,9E+09,9E+09]],
                                        [[-13.7223,784.335,553.685],[0.658015,0.420635,0.529145,0.331796],[-1,1,-2,1],[5156.45,9E+09,9E+09,9E+09,9E+09,9E+09]],
                                        [[-13.71,784.779,554.638],[0.658434,0.420035,0.529448,0.33124],[-1,1,-2,1],[5154.45,9E+09,9E+09,9E+09,9E+09,9E+09]],
                                        [[-13.7037,785.229,555.59],[0.65886,0.419401,0.529775,0.330673],[-1,1,-2,1],[5156.45,9E+09,9E+09,9E+09,9E+09,9E+09]],
                                        [[-13.6974,785.683,556.544],[0.65932,0.418747,0.530101,0.330062],[-1,1,-2,1],[5154.45,9E+09,9E+09,9E+09,9E+09,9E+09]],
                                        [[-13.6915,786.137,557.498],[0.659772,0.418058,0.530456,0.329461],[-1,1,-2,1],[5156.45,9E+09,9E+09,9E+09,9E+09,9E+09]],
                                        [[-13.6815,786.596,558.451],[0.660245,0.417334,0.530823,0.32884],[-1,1,-2,1],[5154.45,9E+09,9E+09,9E+09,9E+09,9E+09]],
                                        [[-13.6731,787.055,559.402],[0.660723,0.416577,0.531214,0.328208],[-1,1,-2,1],[5152.45,9E+09,9E+09,9E+09,9E+09,9E+09]],
                                        [[-13.6624,787.513,560.354],[0.66122,0.415784,0.531623,0.327548],[-1,1,-2,1],[5154.45,9E+09,9E+09,9E+09,9E+09,9E+09]],
                                        [[-13.6531,787.971,561.304],[0.66174,0.414976,0.53203,0.326862],[-1,1,-2,1],[5152.45,9E+09,9E+09,9E+09,9E+09,9E+09]],
                                        [[-13.64,788.437,562.253],[0.662267,0.414159,0.532445,0.326153],[-1,1,-2,1],[5154.45,9E+09,9E+09,9E+09,9E+09,9E+09]],
                                        [[-13.6286,788.904,563.201],[0.662822,0.413305,0.532872,0.325414],[-1,1,-2,1],[5152.45,9E+09,9E+09,9E+09,9E+09,9E+09]],
                                        [[-13.6208,789.377,564.148],[0.663394,0.412414,0.533321,0.324641],[-1,1,-2,1],[5154.45,9E+09,9E+09,9E+09,9E+09,9E+09]],
                                        [[-13.6105,789.852,565.093],[0.664006,0.411501,0.533769,0.323809],[-1,1,-2,1],[5152.45,9E+09,9E+09,9E+09,9E+09,9E+09]],
                                        [[-13.601,790.329,566.038],[0.664603,0.410551,0.534248,0.323001],[-1,1,-2,1],[5154.45,9E+09,9E+09,9E+09,9E+09,9E+09]],
                                        [[-13.59,790.809,566.987],[0.665246,0.40961,0.534698,0.322126],[-1,1,-2,1],[5152.45,9E+09,9E+09,9E+09,9E+09,9E+09]],
                                        [[-13.5816,791.292,567.928],[0.66591,0.408638,0.535166,0.321211],[-1,1,-2,1],[5154.45,9E+09,9E+09,9E+09,9E+09,9E+09]],
                                        [[-13.5754,791.78,568.865],[0.666601,0.407678,0.535604,0.320265],[-1,1,-2,1],[5152.45,9E+09,9E+09,9E+09,9E+09,9E+09]],
                                        [[-13.5693,792.268,569.804],[0.667312,0.406681,0.536063,0.319284],[-1,1,-2,1],[5150.45,9E+09,9E+09,9E+09,9E+09,9E+09]],
                                        [[-13.5606,792.761,570.741],[0.668046,0.405701,0.536495,0.318269],[-1,1,-2,1],[5152.45,9E+09,9E+09,9E+09,9E+09,9E+09]],
                                        [[-13.5486,793.258,571.683],[0.668819,0.404712,0.536913,0.317198],[-1,1,-2,1],[5150.45,9E+09,9E+09,9E+09,9E+09,9E+09]],
                                        [[-13.5339,793.758,572.616],[0.669591,0.403717,0.537335,0.31612],[-1,1,-2,1],[5152.45,9E+09,9E+09,9E+09,9E+09,9E+09]],
                                        [[-13.524,794.259,573.547],[0.670405,0.40271,0.537737,0.314993],[-1,1,-2,1],[5150.45,9E+09,9E+09,9E+09,9E+09,9E+09]],
                                        [[-13.515,794.765,574.479],[0.671222,0.401691,0.538146,0.313854],[-1,1,-2,1],[5152.45,9E+09,9E+09,9E+09,9E+09,9E+09]],
                                        [[-13.5015,795.274,575.415],[0.672076,0.400678,0.538525,0.312669],[-1,1,-2,1],[5154.45,9E+09,9E+09,9E+09,9E+09,9E+09]],
                                        [[-13.4896,795.786,576.344],[0.672932,0.399669,0.538894,0.311481],[-1,1,-2,1],[5152.45,9E+09,9E+09,9E+09,9E+09,9E+09]],
                                        [[-13.4815,796.304,577.272],[0.673796,0.398665,0.539251,0.31028],[-1,1,-2,1],[5154.45,9E+09,9E+09,9E+09,9E+09,9E+09]],
                                        [[-13.4664,796.824,578.195],[0.674667,0.397676,0.539584,0.309075],[-1,1,-2,1],[5152.45,9E+09,9E+09,9E+09,9E+09,9E+09]],
                                        [[-13.4592,797.346,579.111],[0.675559,0.39669,0.539903,0.307834],[-1,1,-2,1],[5154.45,9E+09,9E+09,9E+09,9E+09,9E+09]],
                                        [[-13.4428,797.877,580.038],[0.676453,0.395758,0.540177,0.306587],[-1,1,-2,1],[5152.45,9E+09,9E+09,9E+09,9E+09,9E+09]],
                                        [[-13.4259,798.416,580.953],[0.677359,0.394826,0.540441,0.305321],[-1,1,-2,1],[5154.45,9E+09,9E+09,9E+09,9E+09,9E+09]],
                                        [[-13.4209,798.946,581.868],[0.678267,0.393911,0.540682,0.304058],[-1,1,-2,1],[5156.45,9E+09,9E+09,9E+09,9E+09,9E+09]],
                                        [[-13.4017,799.484,582.784],[0.679181,0.393008,0.540907,0.302782],[-1,1,-2,1],[5154.45,9E+09,9E+09,9E+09,9E+09,9E+09]],
                                        [[-13.3869,800.031,583.702],[0.680093,0.392113,0.541123,0.301508],[-1,1,-2,1],[5156.45,9E+09,9E+09,9E+09,9E+09,9E+09]],
                                        [[-13.3708,800.577,584.622],[0.680983,0.39126,0.541305,0.300277],[-1,1,-2,1],[5158.45,9E+09,9E+09,9E+09,9E+09,9E+09]],
                                        [[-13.3545,801.14,585.552],[0.681891,0.390404,0.541473,0.299025],[-1,1,-2,1],[5156.45,9E+09,9E+09,9E+09,9E+09,9E+09]],
                                        [[-13.3394,801.693,586.464],[0.682766,0.389552,0.541647,0.297823],[-1,1,-2,1],[5158.45,9E+09,9E+09,9E+09,9E+09,9E+09]],
                                        [[-13.323,802.262,587.388],[0.683646,0.388718,0.541791,0.296631],[-1,1,-2,1],[5160.45,9E+09,9E+09,9E+09,9E+09,9E+09]],
                                        [[-13.305,802.824,588.3],[0.684521,0.387897,0.541916,0.295456],[-1,1,-2,1],[5158.45,9E+09,9E+09,9E+09,9E+09,9E+09]],
                                        [[-13.2854,803.401,589.224],[0.685376,0.387096,0.542035,0.294302],[-1,1,-2,1],[5160.45,9E+09,9E+09,9E+09,9E+09,9E+09]],
                                        [[-13.2652,803.973,590.136],[0.686245,0.386301,0.542131,0.293144],[-1,1,-2,1],[5162.45,9E+09,9E+09,9E+09,9E+09,9E+09]],
                                        [[-13.2453,804.547,591.043],[0.687106,0.385498,0.542228,0.292002],[-1,1,-2,1],[5160.45,9E+09,9E+09,9E+09,9E+09,9E+09]],
                                        [[-13.2282,805.117,591.948],[0.687956,0.384712,0.542315,0.290873],[-1,1,-2,1],[5162.45,9E+09,9E+09,9E+09,9E+09,9E+09]],
                                        [[-13.2108,805.698,592.856],[0.688799,0.383943,0.542383,0.289765],[-1,1,-2,1],[5164.45,9E+09,9E+09,9E+09,9E+09,9E+09]],
                                        [[-13.1936,806.277,593.762],[0.689641,0.383157,0.542452,0.288671],[-1,1,-2,1],[5166.45,9E+09,9E+09,9E+09,9E+09,9E+09]],
                                        [[-13.1734,806.862,594.656],[0.69047,0.382388,0.542505,0.287609],[-1,1,-2,1],[5164.45,9E+09,9E+09,9E+09,9E+09,9E+09]],
                                        [[-13.1508,807.448,595.577],[0.691279,0.38157,0.542595,0.286583],[-1,1,-2,1],[5166.45,9E+09,9E+09,9E+09,9E+09,9E+09]],
                                        [[-13.1274,808.042,596.48],[0.692102,0.380753,0.542664,0.285547],[-1,1,-2,1],[5168.45,9E+09,9E+09,9E+09,9E+09,9E+09]],
                                        [[-13.1098,808.64,597.394],[0.69294,0.379928,0.542726,0.284496],[-1,1,-2,1],[5166.45,9E+09,9E+09,9E+09,9E+09,9E+09]],
                                        [[-13.0857,809.239,598.302],[0.693756,0.379052,0.542826,0.283484],[-1,1,-2,1],[5168.45,9E+09,9E+09,9E+09,9E+09,9E+09]],
                                        [[-13.0662,809.835,599.199],[0.694594,0.378153,0.542917,0.282454],[-1,1,-2,1],[5170.45,9E+09,9E+09,9E+09,9E+09,9E+09]],
                                        [[-13.0489,810.424,600.102],[0.695437,0.377255,0.542998,0.281425],[-1,1,-2,1],[5172.45,9E+09,9E+09,9E+09,9E+09,9E+09]],
                                        [[-13.0223,811.027,600.996],[0.696284,0.37632,0.543095,0.280392],[-1,1,-1,1],[5170.45,9E+09,9E+09,9E+09,9E+09,9E+09]],
                                        [[-13.0048,811.625,601.893],[0.697138,0.375357,0.543206,0.279346],[-1,1,-1,1],[5172.45,9E+09,9E+09,9E+09,9E+09,9E+09]],
                                        [[-12.9842,812.231,602.781],[0.698006,0.374371,0.543308,0.278299],[-1,1,-1,1],[5174.45,9E+09,9E+09,9E+09,9E+09,9E+09]],
                                        [[-12.9667,812.845,603.687],[0.698888,0.373333,0.543433,0.277232],[-1,1,-1,1],[5172.45,9E+09,9E+09,9E+09,9E+09,9E+09]],
                                        [[-12.9471,813.447,604.567],[0.69978,0.372261,0.543572,0.276149],[-1,1,-1,1],[5174.45,9E+09,9E+09,9E+09,9E+09,9E+09]],
                                        [[-12.9259,814.067,605.456],[0.700692,0.371177,0.543696,0.27505],[-1,1,-1,1],[5176.45,9E+09,9E+09,9E+09,9E+09,9E+09]],
                                        [[-12.905,814.676,606.328],[0.701627,0.370056,0.543824,0.273921],[-1,1,-1,1],[5174.45,9E+09,9E+09,9E+09,9E+09,9E+09]],
                                        [[-12.8834,815.293,607.203],[0.702565,0.368905,0.543971,0.272776],[-1,1,-1,1],[5176.45,9E+09,9E+09,9E+09,9E+09,9E+09]],
                                        [[-12.8636,815.904,608.069],[0.70352,0.367749,0.544098,0.271621],[-1,1,-1,1],[5178.45,9E+09,9E+09,9E+09,9E+09,9E+09]],
                                        [[-12.8433,816.519,608.929],[0.704486,0.366573,0.544221,0.270458],[-1,1,-1,1],[5176.45,9E+09,9E+09,9E+09,9E+09,9E+09]],
                                        [[-12.8281,817.144,609.802],[0.705446,0.365377,0.544358,0.269295],[-1,1,-1,1],[5178.45,9E+09,9E+09,9E+09,9E+09,9E+09]],
                                        [[-12.8125,817.77,610.666],[0.706434,0.364166,0.544477,0.268103],[-1,1,-1,1],[5180.45,9E+09,9E+09,9E+09,9E+09,9E+09]],
                                        [[-12.7936,818.402,611.522],[0.707431,0.362981,0.544567,0.266896],[-1,1,-1,1],[5182.45,9E+09,9E+09,9E+09,9E+09,9E+09]],
                                        [[-12.7725,819.039,612.386],[0.708455,0.36177,0.54465,0.26565],[-1,1,-1,1],[5180.45,9E+09,9E+09,9E+09,9E+09,9E+09]],
                                        [[-12.7551,819.676,613.244],[0.709473,0.360553,0.544738,0.264404],[-1,1,-1,1],[5182.45,9E+09,9E+09,9E+09,9E+09,9E+09]],
                                        [[-12.7403,820.322,614.084],[0.710521,0.359369,0.544781,0.263111],[-1,1,-1,1],[5184.45,9E+09,9E+09,9E+09,9E+09,9E+09]],
                                        [[-12.719,820.963,614.938],[0.711581,0.358187,0.544805,0.261806],[-1,1,-1,1],[5186.45,9E+09,9E+09,9E+09,9E+09,9E+09]],
                                        [[-12.7015,821.61,615.777],[0.71263,0.357027,0.544812,0.260518],[-1,1,-1,1],[5184.45,9E+09,9E+09,9E+09,9E+09,9E+09]],
                                        [[-12.6808,822.273,616.629],[0.713682,0.355893,0.544798,0.259216],[-1,1,-1,1],[5186.45,9E+09,9E+09,9E+09,9E+09,9E+09]],
                                        [[-12.6646,822.931,617.475],[0.714745,0.354793,0.544741,0.257911],[-1,1,-1,1],[5188.45,9E+09,9E+09,9E+09,9E+09,9E+09]],
                                        [[-12.6458,823.606,618.312],[0.715815,0.35369,0.544676,0.256594],[-1,1,-1,1],[5190.45,9E+09,9E+09,9E+09,9E+09,9E+09]],
                                        [[-12.6264,824.272,619.156],[0.716884,0.352615,0.544581,0.255286],[-1,1,-1,1],[5192.45,9E+09,9E+09,9E+09,9E+09,9E+09]],
                                        [[-12.6094,824.936,619.976],[0.717956,0.351576,0.544453,0.253978],[-1,1,-1,1],[5190.45,9E+09,9E+09,9E+09,9E+09,9E+09]],
                                        [[-12.5926,825.591,620.791],[0.719018,0.35055,0.544319,0.252674],[-1,1,-1,1],[5192.45,9E+09,9E+09,9E+09,9E+09,9E+09]],
                                        [[-12.5734,826.25,621.599],[0.720102,0.349534,0.544151,0.251353],[-1,1,-1,1],[5194.45,9E+09,9E+09,9E+09,9E+09,9E+09]],
                                        [[-12.5545,826.914,622.416],[0.721185,0.348573,0.543942,0.250032],[-1,1,-1,1],[5196.45,9E+09,9E+09,9E+09,9E+09,9E+09]],
                                        [[-12.5371,827.58,623.229],[0.722276,0.34763,0.543707,0.248706],[-1,1,-1,1],[5198.45,9E+09,9E+09,9E+09,9E+09,9E+09]],
                                        [[-12.517,828.255,624.05],[0.723359,0.346705,0.543456,0.247392],[-1,1,-1,1],[5200.45,9E+09,9E+09,9E+09,9E+09,9E+09]],
                                        [[-12.4981,828.946,624.885],[0.724448,0.345801,0.54318,0.246074],[-1,1,-1,1],[5202.45,9E+09,9E+09,9E+09,9E+09,9E+09]],
                                        [[-12.476,829.624,625.706],[0.725549,0.344875,0.542898,0.244748],[-1,1,-1,1],[5204.45,9E+09,9E+09,9E+09,9E+09,9E+09]],
                                        [[-12.4577,830.327,626.523],[0.726642,0.343973,0.542592,0.243449],[-1,1,-1,1],[5206.45,9E+09,9E+09,9E+09,9E+09,9E+09]],
                                        [[-12.4353,831.016,627.328],[0.727728,0.343089,0.542273,0.242158],[-1,1,-1,1],[5208.45,9E+09,9E+09,9E+09,9E+09,9E+09]],
                                        [[-12.4078,831.709,628.147],[0.728829,0.342225,0.541929,0.24084],[-1,1,-1,1],[5210.45,9E+09,9E+09,9E+09,9E+09,9E+09]],
                                        [[-12.3873,832.394,628.955],[0.729941,0.34131,0.541593,0.239522],[-1,1,-1,1],[5212.45,9E+09,9E+09,9E+09,9E+09,9E+09]],
                                        [[-12.3662,833.089,629.751],[0.731031,0.340466,0.541217,0.238244],[-1,1,-1,1],[5214.45,9E+09,9E+09,9E+09,9E+09,9E+09]],
                                        [[-12.3457,833.786,630.565],[0.732138,0.33963,0.540821,0.236933],[-1,1,-1,1],[5216.45,9E+09,9E+09,9E+09,9E+09,9E+09]],
                                        [[-12.3216,834.482,631.367],[0.733248,0.33876,0.540437,0.235621],[-1,1,-1,1],[5218.45,9E+09,9E+09,9E+09,9E+09,9E+09]],
                                        [[-12.301,835.184,632.158],[0.734348,0.337903,0.540038,0.234337],[-1,1,-1,1],[5220.45,9E+09,9E+09,9E+09,9E+09,9E+09]],
                                        [[-12.2779,835.893,632.961],[0.735466,0.337012,0.53964,0.233026],[-1,1,-1,1],[5222.45,9E+09,9E+09,9E+09,9E+09,9E+09]],
                                        [[-12.2543,836.588,633.75],[0.736597,0.336133,0.539222,0.231686],[-1,1,-1,1],[5224.45,9E+09,9E+09,9E+09,9E+09,9E+09]],
                                        [[-12.2321,837.295,634.528],[0.737747,0.335197,0.538816,0.230325],[-1,1,-1,1],[5226.45,9E+09,9E+09,9E+09,9E+09,9E+09]],
                                        [[-12.2114,838.008,635.331],[0.738892,0.334242,0.538411,0.228986],[-1,1,-1,1],[5228.45,9E+09,9E+09,9E+09,9E+09,9E+09]],
                                        [[-12.1853,838.722,636.116],[0.740055,0.333284,0.537992,0.22761],[-1,1,-1,1],[5230.45,9E+09,9E+09,9E+09,9E+09,9E+09]],
                                        [[-12.1626,839.447,636.907],[0.741215,0.332314,0.537569,0.226247],[-1,1,-1,1],[5232.45,9E+09,9E+09,9E+09,9E+09,9E+09]],
                                        [[-12.1418,840.184,637.713],[0.742375,0.331309,0.537152,0.224901],[-1,1,-1,1],[5234.45,9E+09,9E+09,9E+09,9E+09,9E+09]],
                                        [[-12.1133,840.916,638.497],[0.74353,0.33034,0.536712,0.223558],[-1,1,-1,1],[5236.45,9E+09,9E+09,9E+09,9E+09,9E+09]],
                                        [[-12.0913,841.651,639.274],[0.744691,0.329319,0.536284,0.222224],[-1,1,-1,1],[5238.45,9E+09,9E+09,9E+09,9E+09,9E+09]],
                                        [[-12.0727,842.392,640.061],[0.745841,0.328313,0.535844,0.220915],[-1,1,-1,1],[5240.45,9E+09,9E+09,9E+09,9E+09,9E+09]],
                                        [[-12.0499,843.134,640.848],[0.747001,0.327296,0.535397,0.219584],[-1,1,-1,1],[5242.45,9E+09,9E+09,9E+09,9E+09,9E+09]],
                                        [[-12.0164,843.864,641.612],[0.74817,0.326232,0.534959,0.218252],[-1,1,-1,1],[5244.45,9E+09,9E+09,9E+09,9E+09,9E+09]],
                                        [[-11.9994,844.609,642.37],[0.74933,0.325187,0.534506,0.216939],[-1,1,-1,1],[5246.45,9E+09,9E+09,9E+09,9E+09,9E+09]],
                                        [[-11.9764,845.343,643.159],[0.7505,0.324124,0.534048,0.215608],[-1,1,-1,1],[5248.45,9E+09,9E+09,9E+09,9E+09,9E+09]],
                                        [[-11.9415,846.088,643.927],[0.751685,0.323054,0.533579,0.214243],[-1,1,-1,1],[5250.45,9E+09,9E+09,9E+09,9E+09,9E+09]],
                                        [[-11.9236,846.837,644.677],[0.752859,0.321946,0.533124,0.212914],[-1,1,-1,1],[5252.45,9E+09,9E+09,9E+09,9E+09,9E+09]],
                                        [[-11.9013,847.599,645.455],[0.754026,0.320866,0.532651,0.211595],[-1,1,-1,1],[5254.45,9E+09,9E+09,9E+09,9E+09,9E+09]],
                                        [[-11.8746,848.372,646.235],[0.755208,0.319749,0.532179,0.210256],[-1,1,-1,1],[5256.45,9E+09,9E+09,9E+09,9E+09,9E+09]],
                                        [[-11.8397,849.142,646.989],[0.75638,0.318629,0.531702,0.208947],[-1,1,-1,1],[5258.45,9E+09,9E+09,9E+09,9E+09,9E+09]],
                                        [[-11.8171,849.907,647.734],[0.757556,0.317508,0.531212,0.207633],[-1,1,-1,1],[5260.45,9E+09,9E+09,9E+09,9E+09,9E+09]],
                                        [[-11.7978,850.683,648.499],[0.758742,0.316368,0.530717,0.206306],[-1,1,-1,1],[5262.45,9E+09,9E+09,9E+09,9E+09,9E+09]],
                                        [[-11.7622,851.449,649.242],[0.759913,0.315245,0.530208,0.205018],[-1,1,-1,1],[5264.45,9E+09,9E+09,9E+09,9E+09,9E+09]],
                                        [[-11.741,852.221,649.984],[0.761085,0.314103,0.529696,0.203744],[-1,1,-1,1],[5266.45,9E+09,9E+09,9E+09,9E+09,9E+09]],
                                        [[-11.7225,853.004,650.744],[0.762262,0.312997,0.529154,0.202446],[-1,1,-1,1],[5268.45,9E+09,9E+09,9E+09,9E+09,9E+09]],
                                        [[-11.69,853.77,651.483],[0.763444,0.311876,0.528606,0.201151],[-1,1,-1,1],[5270.45,9E+09,9E+09,9E+09,9E+09,9E+09]],
                                        [[-11.6729,854.551,652.222],[0.764616,0.310759,0.528048,0.19989],[-1,1,-1,1],[5272.45,9E+09,9E+09,9E+09,9E+09,9E+09]],
                                        [[-11.6517,855.344,652.977],[0.76579,0.309644,0.527477,0.198632],[-1,1,-1,1],[5274.45,9E+09,9E+09,9E+09,9E+09,9E+09]],
                                        [[-11.6178,856.126,653.708],[0.766962,0.30854,0.526889,0.197381],[-1,1,-1,1],[5276.45,9E+09,9E+09,9E+09,9E+09,9E+09]],
                                        [[-11.6009,856.917,654.433],[0.768134,0.307425,0.526299,0.196138],[-1,1,-1,1],[5278.45,9E+09,9E+09,9E+09,9E+09,9E+09]],
                                        [[-11.5821,857.71,655.176],[0.769312,0.306354,0.52568,0.194852],[-1,1,-1,1],[5280.45,9E+09,9E+09,9E+09,9E+09,9E+09]],
                                        [[-11.5528,858.518,655.91],[0.770506,0.305235,0.525069,0.193534],[-1,1,-1,1],[5282.45,9E+09,9E+09,9E+09,9E+09,9E+09]],
                                        [[-11.5185,859.312,656.617],[0.771677,0.304155,0.524443,0.192261],[-1,1,-1,1],[5284.45,9E+09,9E+09,9E+09,9E+09,9E+09]],
                                        [[-11.5069,860.109,657.326],[0.772853,0.30311,0.523794,0.190951],[-1,1,-1,1],[5286.45,9E+09,9E+09,9E+09,9E+09,9E+09]],
                                        [[-11.4799,860.908,658.057],[0.77404,0.30204,0.523145,0.189615],[-1,1,-1,1],[5288.45,9E+09,9E+09,9E+09,9E+09,9E+09]],
                                        [[-11.4534,861.723,658.771],[0.775222,0.300974,0.52249,0.188283],[-1,1,-1,1],[5290.45,9E+09,9E+09,9E+09,9E+09,9E+09]],
                                        [[-11.4377,862.527,659.48],[0.77639,0.299919,0.521829,0.18698],[-1,1,-1,1],[5292.45,9E+09,9E+09,9E+09,9E+09,9E+09]],
                                        [[-11.4121,863.344,660.192],[0.777571,0.298871,0.521154,0.185629],[-1,1,-1,1],[5294.45,9E+09,9E+09,9E+09,9E+09,9E+09]],
                                        [[-11.3866,864.146,660.891],[0.778762,0.297803,0.520476,0.184248],[-1,1,-1,1],[5296.45,9E+09,9E+09,9E+09,9E+09,9E+09]],
                                        [[-11.3669,864.955,661.588],[0.779944,0.296744,0.519792,0.182885],[-1,1,-1,1],[5298.45,9E+09,9E+09,9E+09,9E+09,9E+09]],
                                        [[-11.3532,865.773,662.297],[0.781131,0.295689,0.519098,0.181493],[-1,1,-1,1],[5300.45,9E+09,9E+09,9E+09,9E+09,9E+09]],
                                        [[-11.3148,866.592,663.001],[0.782318,0.294626,0.5184,0.180098],[-1,1,-1,1],[5302.45,9E+09,9E+09,9E+09,9E+09,9E+09]],
                                        [[-11.2903,867.399,663.676],[0.783498,0.29356,0.517701,0.178717],[-1,1,-1,1],[5304.45,9E+09,9E+09,9E+09,9E+09,9E+09]],
                                        [[-11.2804,868.211,664.374],[0.784676,0.292531,0.51698,0.177317],[-1,1,-1,1],[5306.45,9E+09,9E+09,9E+09,9E+09,9E+09]],
                                        [[-11.2549,869.039,665.075],[0.785847,0.291502,0.516256,0.175927],[-1,1,-1,1],[5308.45,9E+09,9E+09,9E+09,9E+09,9E+09]],
                                        [[-11.2258,869.863,665.766],[0.786999,0.290474,0.515534,0.174593],[-1,1,-1,1],[5310.45,9E+09,9E+09,9E+09,9E+09,9E+09]],
                                        [[-11.2033,870.7,666.452],[0.788147,0.289485,0.514792,0.173242],[-1,1,-1,1],[5312.45,9E+09,9E+09,9E+09,9E+09,9E+09]],
                                        [[-11.1667,871.541,667.144],[0.789295,0.288476,0.514051,0.171891],[-1,1,-1,1],[5314.45,9E+09,9E+09,9E+09,9E+09,9E+09]],
                                        [[-11.1333,872.378,667.819],[0.790435,0.287465,0.513309,0.170558],[-1,1,-1,1],[5316.45,9E+09,9E+09,9E+09,9E+09,9E+09]],
                                        [[-11.1111,873.224,668.498],[0.791574,0.286465,0.512557,0.169214],[-1,1,-1,1],[5318.45,9E+09,9E+09,9E+09,9E+09,9E+09]],
                                        [[-11.0774,874.07,669.182],[0.792721,0.285448,0.511802,0.167843],[-1,1,-1,1],[5320.45,9E+09,9E+09,9E+09,9E+09,9E+09]],
                                        [[-11.0417,874.917,669.845],[0.79386,0.284382,0.511064,0.166513],[-1,1,-1,1],[5322.45,9E+09,9E+09,9E+09,9E+09,9E+09]],
                                        [[-11.0126,875.751,670.502],[0.794981,0.283346,0.510317,0.165218],[-1,1,-1,1],[5324.45,9E+09,9E+09,9E+09,9E+09,9E+09]],
                                        [[-10.9928,876.601,671.172],[0.796107,0.28228,0.509573,0.163912],[-1,1,-1,1],[5326.45,9E+09,9E+09,9E+09,9E+09,9E+09]],
                                        [[-10.9603,877.455,671.844],[0.797215,0.281197,0.508838,0.162668],[-1,1,-1,1],[5328.45,9E+09,9E+09,9E+09,9E+09,9E+09]],
                                        [[-10.9262,878.309,672.495],[0.798326,0.280073,0.508112,0.161421],[-1,1,-1,1],[5330.45,9E+09,9E+09,9E+09,9E+09,9E+09]],
                                        [[-10.8961,879.158,673.142],[0.799423,0.278977,0.507376,0.160203],[-1,1,-1,1],[5332.45,9E+09,9E+09,9E+09,9E+09,9E+09]],
                                        [[-10.8695,880.019,673.8],[0.800516,0.277848,0.506648,0.159003],[-1,1,-1,1],[5334.45,9E+09,9E+09,9E+09,9E+09,9E+09]],
                                        [[-10.8383,880.881,674.458],[0.801595,0.276704,0.505927,0.157853],[-1,1,-1,1],[5336.45,9E+09,9E+09,9E+09,9E+09,9E+09]],
                                        [[-10.8075,881.748,675.104],[0.80267,0.275573,0.505197,0.156705],[-1,1,-1,1],[5338.45,9E+09,9E+09,9E+09,9E+09,9E+09]],
                                        [[-10.7738,882.597,675.743],[0.803742,0.274421,0.50447,0.155566],[-1,1,-1,1],[5340.45,9E+09,9E+09,9E+09,9E+09,9E+09]],
                                        [[-10.7401,883.444,676.376],[0.804795,0.273271,0.503747,0.154489],[-1,1,-1,1],[5342.45,9E+09,9E+09,9E+09,9E+09,9E+09]],
                                        [[-10.7227,884.307,677.021],[0.805836,0.272124,0.503022,0.153448],[-1,1,-1,1],[5344.45,9E+09,9E+09,9E+09,9E+09,9E+09]],
                                        [[-10.6896,885.174,677.671],[0.806869,0.270981,0.502294,0.152424],[-1,1,-1,1],[5346.45,9E+09,9E+09,9E+09,9E+09,9E+09]],
                                        [[-10.655,886.046,678.304],[0.807898,0.269792,0.501579,0.151431],[-1,1,-1,1],[5348.45,9E+09,9E+09,9E+09,9E+09,9E+09]],
                                        [[-10.6231,886.92,678.93],[0.80893,0.268585,0.500864,0.150431],[-1,1,-1,1],[5350.45,9E+09,9E+09,9E+09,9E+09,9E+09]],
                                        [[-10.5905,887.792,679.551],[0.809968,0.267349,0.500151,0.149417],[-1,1,-1,1],[5352.45,9E+09,9E+09,9E+09,9E+09,9E+09]],
                                        [[-10.564,888.659,680.173],[0.811003,0.266077,0.499447,0.148424],[-1,1,-1,1],[5354.45,9E+09,9E+09,9E+09,9E+09,9E+09]],
                                        [[-10.5415,889.532,680.789],[0.812042,0.264781,0.498743,0.147426],[-1,1,-1,1],[5356.45,9E+09,9E+09,9E+09,9E+09,9E+09]],
                                        [[-10.517,890.402,681.404],[0.813085,0.263472,0.498036,0.14641],[-1,1,-1,1],[5358.45,9E+09,9E+09,9E+09,9E+09,9E+09]],
                                        [[-10.489,891.274,682.015],[0.814133,0.262116,0.497337,0.145392],[-1,1,-1,1],[5360.45,9E+09,9E+09,9E+09,9E+09,9E+09]],
                                        [[-10.4711,892.154,682.626],[0.815175,0.260727,0.496647,0.144409],[-1,1,-1,1],[5362.45,9E+09,9E+09,9E+09,9E+09,9E+09]],
                                        [[-10.4466,893.035,683.235],[0.816216,0.259325,0.495955,0.143427],[-1,1,-1,1],[5364.45,9E+09,9E+09,9E+09,9E+09,9E+09]],
                                        [[-10.4197,893.911,683.84],[0.817263,0.257894,0.495263,0.142428],[-1,1,-1,1],[5366.45,9E+09,9E+09,9E+09,9E+09,9E+09]],
                                        [[-10.3948,894.794,684.441],[0.818312,0.256436,0.494574,0.141433],[-1,1,-1,1],[5368.45,9E+09,9E+09,9E+09,9E+09,9E+09]],
                                        [[-10.37,895.68,685.04],[0.819356,0.254981,0.493878,0.140443],[-1,1,-1,1],[5370.45,9E+09,9E+09,9E+09,9E+09,9E+09]],
                                        [[-10.3491,896.567,685.636],[0.820406,0.253502,0.493181,0.139436],[-1,1,-1,1],[5372.45,9E+09,9E+09,9E+09,9E+09,9E+09]],
                                        [[-10.3252,897.452,686.232],[0.821454,0.25202,0.492479,0.138432],[-1,1,-1,1],[5374.45,9E+09,9E+09,9E+09,9E+09,9E+09]],
                                        [[-10.2975,898.339,686.821],[0.82251,0.250515,0.491774,0.137397],[-1,1,-1,1],[5376.45,9E+09,9E+09,9E+09,9E+09,9E+09]],
                                        [[-10.2764,899.226,687.407],[0.82356,0.249031,0.491057,0.136365],[-1,1,-1,1],[5378.45,9E+09,9E+09,9E+09,9E+09,9E+09]],
                                        [[-10.2536,900.117,687.99],[0.82461,0.247517,0.490343,0.135344],[-1,1,-1,1],[5380.45,9E+09,9E+09,9E+09,9E+09,9E+09]],
                                        [[-10.2371,901.025,688.569],[0.825657,0.24601,0.489621,0.134316],[-1,1,-1,1],[5382.45,9E+09,9E+09,9E+09,9E+09,9E+09]],
                                        [[-10.2191,901.939,689.144],[0.826706,0.244502,0.488891,0.133272],[-1,1,-1,1],[5384.45,9E+09,9E+09,9E+09,9E+09,9E+09]],
                                        [[-10.1985,902.848,689.714],[0.827757,0.242996,0.488152,0.13221],[-1,1,-1,1],[5386.45,9E+09,9E+09,9E+09,9E+09,9E+09]],
                                        [[-10.1793,903.767,690.282],[0.828814,0.241476,0.487406,0.131119],[-1,1,-1,1],[5388.45,9E+09,9E+09,9E+09,9E+09,9E+09]],
                                        [[-10.1612,904.688,690.846],[0.829869,0.239963,0.486652,0.13002],[-1,1,-1,1],[5390.45,9E+09,9E+09,9E+09,9E+09,9E+09]],
                                        [[-10.1405,905.602,691.408],[0.830919,0.238448,0.485894,0.128929],[-1,1,-1,1],[5392.45,9E+09,9E+09,9E+09,9E+09,9E+09]],
                                        [[-10.1257,906.52,691.966],[0.831969,0.236925,0.485131,0.127833],[-1,1,-1,1],[5394.45,9E+09,9E+09,9E+09,9E+09,9E+09]],
                                        [[-10.1109,907.451,692.52],[0.833017,0.235414,0.484358,0.126726],[-1,1,-1,1],[5396.45,9E+09,9E+09,9E+09,9E+09,9E+09]],
                                        [[-10.0951,908.375,693.071],[0.834061,0.233892,0.483584,0.125631],[-1,1,-1,1],[5398.45,9E+09,9E+09,9E+09,9E+09,9E+09]],
                                        [[-10.0786,909.301,693.62],[0.835097,0.232386,0.482802,0.124547],[-1,1,-1,1],[5400.45,9E+09,9E+09,9E+09,9E+09,9E+09]],
                                        [[-10.0657,910.23,694.167],[0.836132,0.230889,0.48201,0.123451],[-1,1,-1,1],[5402.45,9E+09,9E+09,9E+09,9E+09,9E+09]],
                                        [[-10.0449,911.161,694.71],[0.837162,0.229408,0.481209,0.122351],[-1,1,-1,1],[5404.45,9E+09,9E+09,9E+09,9E+09,9E+09]],
                                        [[-10.0267,912.092,695.253],[0.838191,0.227931,0.480399,0.121242],[-1,1,-1,1],[5406.45,9E+09,9E+09,9E+09,9E+09,9E+09]],
                                        [[-10.0115,913.029,695.788],[0.839215,0.226464,0.479583,0.120136],[-1,1,-1,1],[5408.45,9E+09,9E+09,9E+09,9E+09,9E+09]],
                                        [[-9.9934,913.969,696.323],[0.840236,0.225011,0.478757,0.119019],[-1,1,-1,1],[5410.45,9E+09,9E+09,9E+09,9E+09,9E+09]],
                                        [[-9.97878,914.911,696.855],[0.841245,0.22361,0.477914,0.117911],[-1,1,-1,1],[5412.45,9E+09,9E+09,9E+09,9E+09,9E+09]],
                                        [[-9.96001,915.857,697.384],[0.842255,0.222194,0.47707,0.116798],[-1,1,-1,1],[5414.45,9E+09,9E+09,9E+09,9E+09,9E+09]],
                                        [[-9.94509,916.805,697.905],[0.843255,0.220799,0.476217,0.115697],[-1,1,-1,1],[5416.45,9E+09,9E+09,9E+09,9E+09,9E+09]],
                                        [[-9.93088,917.761,698.427],[0.844248,0.219402,0.475363,0.11462],[-1,1,-1,1],[5418.34,9E+09,9E+09,9E+09,9E+09,9E+09]],
                                        [[-9.91375,918.719,698.949],[0.845239,0.218001,0.474505,0.113539],[-1,1,-1,1],[5420.11,9E+09,9E+09,9E+09,9E+09,9E+09]],
                                        [[-9.89736,919.68,699.464],[0.84623,0.216583,0.473646,0.112455],[-1,1,-1,1],[5421.77,9E+09,9E+09,9E+09,9E+09,9E+09]],
                                        [[-9.8792,920.636,699.976],[0.847215,0.215174,0.472781,0.111379],[-1,1,-1,1],[5423.31,9E+09,9E+09,9E+09,9E+09,9E+09]],
                                        [[-9.8647,921.592,700.486],[0.848203,0.213731,0.471917,0.110293],[-1,1,-1,1],[5424.75,9E+09,9E+09,9E+09,9E+09,9E+09]],
                                        [[-9.84857,922.555,700.991],[0.84918,0.212326,0.471042,0.109223],[-1,1,-1,1],[5426.07,9E+09,9E+09,9E+09,9E+09,9E+09]],
                                        [[-9.83135,923.513,701.491],[0.850157,0.2109,0.470168,0.108153],[-1,1,-1,1],[5427.26,9E+09,9E+09,9E+09,9E+09,9E+09]],
                                        [[-9.81631,924.47,701.987],[0.851135,0.209442,0.469295,0.107081],[-1,1,-1,1],[5428.35,9E+09,9E+09,9E+09,9E+09,9E+09]],
                                        [[-9.80313,925.437,702.482],[0.852107,0.207985,0.468418,0.106018],[-1,1,-1,1],[5429.32,9E+09,9E+09,9E+09,9E+09,9E+09]],
                                        [[-9.78621,926.407,702.972],[0.853079,0.206514,0.46754,0.104954],[-1,1,-1,1],[5430.17,9E+09,9E+09,9E+09,9E+09,9E+09]],
                                        [[-9.76926,927.367,703.458],[0.854043,0.205047,0.466658,0.103908],[-1,1,-1,1],[5430.89,9E+09,9E+09,9E+09,9E+09,9E+09]],
                                        [[-9.75267,928.338,703.941],[0.855007,0.203571,0.465772,0.102854],[-1,1,-1,1],[5431.5,9E+09,9E+09,9E+09,9E+09,9E+09]],
                                        [[-9.73612,929.311,704.419],[0.855966,0.202104,0.46488,0.101799],[-1,1,-1,1],[5431.99,9E+09,9E+09,9E+09,9E+09,9E+09]],
                                        [[-9.71729,930.285,704.895],[0.856925,0.200624,0.463985,0.100739],[-1,1,-1,1],[5432.35,9E+09,9E+09,9E+09,9E+09,9E+09]],
                                        [[-9.70202,931.26,705.367],[0.857875,0.199165,0.463083,0.0996935],[-1,1,-1,1],[5432.59,9E+09,9E+09,9E+09,9E+09,9E+09]],
                                        [[-9.68892,932.237,705.837],[0.858822,0.1977,0.462177,0.0986469],[-1,1,-1,1],[5432.71,9E+09,9E+09,9E+09,9E+09,9E+09]],
                                        [[-9.6772,933.217,706.302],[0.859765,0.196241,0.461267,0.0976028],[-1,1,-1,1],[5432.7,9E+09,9E+09,9E+09,9E+09,9E+09]],
                                        [[-9.66783,934.201,706.763],[0.860704,0.194778,0.460353,0.0965675],[-1,1,-1,1],[5432.57,9E+09,9E+09,9E+09,9E+09,9E+09]],
                                        [[-9.6509,935.181,707.222],[0.86164,0.193308,0.459437,0.0955321],[-1,1,-1,1],[5432.31,9E+09,9E+09,9E+09,9E+09,9E+09]],
                                        [[-9.64026,936.169,707.678],[0.862576,0.191825,0.458517,0.0944898],[-1,1,-1,1],[5431.94,9E+09,9E+09,9E+09,9E+09,9E+09]],
                                        [[-9.62708,937.159,708.131],[0.863506,0.19035,0.457592,0.0934504],[-1,1,-1,1],[5431.43,9E+09,9E+09,9E+09,9E+09,9E+09]],
                                        [[-9.61484,938.15,708.581],[0.864433,0.188883,0.456661,0.0924081],[-1,1,-1,1],[5430.79,9E+09,9E+09,9E+09,9E+09,9E+09]],
                                        [[-9.60129,939.138,709.024],[0.865357,0.187409,0.455727,0.0913663],[-1,1,-1,1],[5430.03,9E+09,9E+09,9E+09,9E+09,9E+09]],
                                        [[-9.58817,940.134,709.467],[0.866275,0.185945,0.454788,0.0903301],[-1,1,-1,1],[5429.15,9E+09,9E+09,9E+09,9E+09,9E+09]],
                                        [[-9.5753,941.127,709.902],[0.867188,0.184485,0.453844,0.0893026],[-1,1,-1,1],[5428.13,9E+09,9E+09,9E+09,9E+09,9E+09]],
                                        [[-9.56211,942.129,710.335],[0.868096,0.183027,0.452898,0.0882852],[-1,1,-1,1],[5426.99,9E+09,9E+09,9E+09,9E+09,9E+09]],
                                        [[-9.54904,943.123,710.765],[0.868999,0.18157,0.451947,0.0872734],[-1,1,-1,1],[5425.71,9E+09,9E+09,9E+09,9E+09,9E+09]],
                                        [[-9.53567,944.121,711.19],[0.869898,0.180117,0.450992,0.0862631],[-1,1,-1,1],[5424.32,9E+09,9E+09,9E+09,9E+09,9E+09]],
                                        [[-9.52331,945.12,711.61],[0.870793,0.178672,0.450032,0.0852521],[-1,1,-1,1],[5422.79,9E+09,9E+09,9E+09,9E+09,9E+09]],
                                        [[-9.50843,946.121,712.025],[0.871683,0.177237,0.449065,0.0842402],[-1,1,-1,1],[5421.14,9E+09,9E+09,9E+09,9E+09,9E+09]],
                                        [[-9.49316,947.119,712.44],[0.872569,0.175807,0.448094,0.0832256],[-1,1,-1,1],[5419.35,9E+09,9E+09,9E+09,9E+09,9E+09]],
                                        [[-9.48088,948.121,712.852],[0.873452,0.174377,0.447119,0.0822138],[-1,1,-1,1],[5417.45,9E+09,9E+09,9E+09,9E+09,9E+09]],
                                        [[-9.46535,949.125,713.261],[0.874329,0.172957,0.446139,0.0812079],[-1,1,-1,1],[5415.45,9E+09,9E+09,9E+09,9E+09,9E+09]],
                                        [[-9.45291,950.131,713.667],[0.875201,0.171538,0.445156,0.0802149],[-1,1,-1,1],[5413.45,9E+09,9E+09,9E+09,9E+09,9E+09]],
                                        [[-9.44121,951.138,714.069],[0.876062,0.170137,0.444171,0.0792521],[-1,1,-1,1],[5411.45,9E+09,9E+09,9E+09,9E+09,9E+09]],
